LIN {X -112.034,Y -13.899,Z -33.351,A -90.000,B 90.000,C 0.000} C_DIS
LIN {X -111.882,Y -13.901,Z -33.215,A -90.000,B 90.000,C 0.000} C_DIS
LIN {X -111.725,Y -13.904,Z -33.072,A -90.000,B 90.000,C 0.000} C_DIS
LIN {X -111.571,Y -13.911,Z -32.939,A -90.000,B 90.000,C 0.000} C_DIS
LIN {X -111.426,Y -13.925,Z -32.809,A -90.000,B 90.000,C 0.000} C_DIS
LIN {X -111.312,Y -13.944,Z -32.695,A -90.000,B 90.000,C 0.000} C_DIS
LIN {X -110.883,Y -13.954,Z -32.137,A -90.000,B 90.000,C 0.000} C_DIS
LIN {X -110.737,Y -13.959,Z -31.950,A -90.000,B 90.000,C 0.000} C_DIS
LIN {X -110.627,Y -13.962,Z -31.815,A -90.000,B 90.000,C 0.000} C_DIS
LIN {X -110.356,Y -13.969,Z -31.490,A -90.000,B 90.000,C 0.000} C_DIS
LIN {X -110.187,Y -13.968,Z -31.297,A -90.000,B 90.000,C 0.000} C_DIS
LIN {X -110.090,Y -13.970,Z -31.191,A -90.000,B 90.000,C 0.000} C_DIS
LIN {X -109.713,Y -13.983,Z -30.801,A -90.000,B 90.000,C 0.000} C_DIS
LIN {X -109.313,Y -13.994,Z -30.426,A -90.000,B 90.000,C 0.000} C_DIS
LIN {X -108.942,Y -13.995,Z -30.095,A -90.000,B 90.000,C 0.000} C_DIS
LIN {X -108.599,Y -14.004,Z -29.802,A -90.000,B 90.000,C 0.000} C_DIS
LIN {X -108.444,Y -14.007,Z -29.672,A -90.000,B 90.000,C 0.000} C_DIS
LIN {X -108.225,Y -14.011,Z -29.494,A -90.000,B 90.000,C 0.000} C_DIS
LIN {X -107.679,Y -14.018,Z -29.057,A -90.000,B 90.000,C 0.000} C_DIS
LIN {X -107.487,Y -14.013,Z -28.912,A -90.000,B 90.000,C 0.000} C_DIS
LIN {X -107.181,Y -14.012,Z -28.694,A -90.000,B 90.000,C 0.000} C_DIS
LIN {X -106.850,Y -14.010,Z -28.465,A -90.000,B 90.000,C 0.000} C_DIS
LIN {X -106.554,Y -13.995,Z -28.277,A -90.000,B 90.000,C 0.000} C_DIS
LIN {X -106.262,Y -13.993,Z -28.107,A -90.000,B 90.000,C 0.000} C_DIS
LIN {X -105.912,Y -13.982,Z -27.915,A -90.000,B 90.000,C 0.000} C_DIS
LIN {X -105.604,Y -13.971,Z -27.766,A -90.000,B 90.000,C 0.000} C_DIS
LIN {X -105.412,Y -13.966,Z -27.676,A -90.000,B 90.000,C 0.000} C_DIS
LIN {X -105.178,Y -13.965,Z -27.574,A -90.000,B 90.000,C 0.000} C_DIS
LIN {X -104.756,Y -13.950,Z -27.404,A -90.000,B 90.000,C 0.000} C_DIS
LIN {X -104.528,Y -13.941,Z -27.320,A -90.000,B 90.000,C 0.000} C_DIS
LIN {X -104.102,Y -13.933,Z -27.170,A -90.000,B 90.000,C 0.000} C_DIS
LIN {X -103.873,Y -13.933,Z -27.095,A -90.000,B 90.000,C 0.000} C_DIS
LIN {X -103.252,Y -13.916,Z -26.894,A -90.000,B 90.000,C 0.000} C_DIS
LIN {X -102.946,Y -13.913,Z -26.800,A -90.000,B 90.000,C 0.000} C_DIS
LIN {X -102.732,Y -13.819,Z -26.639,A -90.000,B 90.000,C 0.000} C_DIS
LIN {X -102.589,Y -13.762,Z -26.537,A -90.000,B 90.000,C 0.000} C_DIS
LIN {X -102.458,Y -13.716,Z -26.450,A -90.000,B 90.000,C 0.000} C_DIS
LIN {X -102.318,Y -13.669,Z -26.360,A -90.000,B 90.000,C 0.000} C_DIS
LIN {X -102.306,Y -13.670,Z -26.341,A -90.000,B 90.000,C 0.000} C_DIS
LIN {X -102.042,Y -13.676,Z -25.951,A -90.000,B 90.000,C 0.000} C_DIS
LIN {X -101.875,Y -13.681,Z -25.720,A -90.000,B 90.000,C 0.000} C_DIS
LIN {X -101.706,Y -13.682,Z -25.502,A -90.000,B 90.000,C 0.000} C_DIS
LIN {X -101.671,Y -13.685,Z -25.450,A -90.000,B 90.000,C 0.000} C_DIS
LIN {X -101.467,Y -13.684,Z -25.192,A -90.000,B 90.000,C 0.000} C_DIS
LIN {X -101.393,Y -13.692,Z -25.087,A -90.000,B 90.000,C 0.000} C_DIS
LIN {X -101.277,Y -13.697,Z -24.936,A -90.000,B 90.000,C 0.000} C_DIS
LIN {X -101.079,Y -13.713,Z -24.676,A -90.000,B 90.000,C 0.000} C_DIS
LIN {X -100.863,Y -13.726,Z -24.406,A -90.000,B 90.000,C 0.000} C_DIS
LIN {X -100.744,Y -13.738,Z -24.262,A -90.000,B 90.000,C 0.000} C_DIS
LIN {X -100.655,Y -13.743,Z -24.163,A -90.000,B 90.000,C 0.000} C_DIS
LIN {X -100.615,Y -13.744,Z -24.116,A -90.000,B 90.000,C 0.000} C_DIS
LIN {X -100.507,Y -13.750,Z -23.996,A -90.000,B 90.000,C 0.000} C_DIS
LIN {X -100.359,Y -13.763,Z -23.838,A -90.000,B 90.000,C 0.000} C_DIS
LIN {X -100.223,Y -13.773,Z -23.695,A -90.000,B 90.000,C 0.000} C_DIS
LIN {X -99.934,Y -13.779,Z -23.429,A -90.000,B 90.000,C 0.000} C_DIS
LIN {X -99.843,Y -13.783,Z -23.348,A -90.000,B 90.000,C 0.000} C_DIS
LIN {X -99.649,Y -13.788,Z -23.183,A -90.000,B 90.000,C 0.000} C_DIS
LIN {X -99.518,Y -13.792,Z -23.082,A -90.000,B 90.000,C 0.000} C_DIS
LIN {X -99.172,Y -13.792,Z -22.838,A -90.000,B 90.000,C 0.000} C_DIS
LIN {X -98.955,Y -13.787,Z -22.696,A -90.000,B 90.000,C 0.000} C_DIS
LIN {X -98.690,Y -13.777,Z -22.542,A -90.000,B 90.000,C 0.000} C_DIS
LIN {X -98.581,Y -13.777,Z -22.483,A -90.000,B 90.000,C 0.000} C_DIS
LIN {X -98.305,Y -13.760,Z -22.357,A -90.000,B 90.000,C 0.000} C_DIS
LIN {X -98.201,Y -13.756,Z -22.312,A -90.000,B 90.000,C 0.000} C_DIS
LIN {X -98.005,Y -13.745,Z -22.237,A -90.000,B 90.000,C 0.000} C_DIS
LIN {X -97.903,Y -13.741,Z -22.200,A -90.000,B 90.000,C 0.000} C_DIS
LIN {X -97.496,Y -13.717,Z -22.072,A -90.000,B 90.000,C 0.000} C_DIS
LIN {X -97.397,Y -13.709,Z -22.050,A -90.000,B 90.000,C 0.000} C_DIS
LIN {X -97.037,Y -13.687,Z -21.979,A -90.000,B 90.000,C 0.000} C_DIS
LIN {X -96.920,Y -13.678,Z -21.961,A -90.000,B 90.000,C 0.000} C_DIS
LIN {X -96.713,Y -13.661,Z -21.934,A -90.000,B 90.000,C 0.000} C_DIS
LIN {X -96.487,Y -13.648,Z -21.909,A -90.000,B 90.000,C 0.000} C_DIS
LIN {X -96.193,Y -13.619,Z -21.899,A -90.000,B 90.000,C 0.000} C_DIS
LIN {X -96.028,Y -13.611,Z -21.893,A -90.000,B 90.000,C 0.000} C_DIS
LIN {X -95.877,Y -13.604,Z -21.893,A -90.000,B 90.000,C 0.000} C_DIS
LIN {X -95.614,Y -13.584,Z -21.906,A -90.000,B 90.000,C 0.000} C_DIS
LIN {X -95.537,Y -13.622,Z -21.843,A -90.000,B 90.000,C 0.000} C_DIS
LIN {X -95.434,Y -13.674,Z -21.767,A -90.000,B 90.000,C 0.000} C_DIS
LIN {X -95.337,Y -13.724,Z -21.703,A -90.000,B 90.000,C 0.000} C_DIS
LIN {X -95.205,Y -13.792,Z -21.624,A -90.000,B 90.000,C 0.000} C_DIS
LIN {X -95.067,Y -13.866,Z -21.548,A -90.000,B 90.000,C 0.000} C_DIS
LIN {X -94.996,Y -13.904,Z -21.514,A -90.000,B 90.000,C 0.000} C_DIS
LIN {X -94.934,Y -13.938,Z -21.487,A -90.000,B 90.000,C 0.000} C_DIS
LIN {X -94.872,Y -13.972,Z -21.461,A -90.000,B 90.000,C 0.000} C_DIS
LIN {X -94.732,Y -14.044,Z -21.414,A -90.000,B 90.000,C 0.000} C_DIS
LIN {X -94.570,Y -14.126,Z -21.368,A -90.000,B 90.000,C 0.000} C_DIS
LIN {X -94.236,Y -14.315,Z -21.280,A -90.000,B 90.000,C 0.000} C_DIS
LIN {X -94.158,Y -14.359,Z -21.266,A -90.000,B 90.000,C 0.000} C_DIS
LIN {X -94.070,Y -14.402,Z -21.258,A -90.000,B 90.000,C 0.000} C_DIS
LIN {X -93.862,Y -14.506,Z -21.250,A -90.000,B 90.000,C 0.000} C_DIS
LIN {X -93.860,Y -14.506,Z -21.241,A -90.000,B 90.000,C 0.000} C_DIS
LIN {X -93.780,Y -14.481,Z -20.924,A -90.000,B 90.000,C 0.000} C_DIS
LIN {X -93.747,Y -14.467,Z -20.815,A -90.000,B 90.000,C 0.000} C_DIS
LIN {X -93.701,Y -14.454,Z -20.689,A -90.000,B 90.000,C 0.000} C_DIS
LIN {X -93.679,Y -14.449,Z -20.634,A -90.000,B 90.000,C 0.000} C_DIS
LIN {X -93.611,Y -14.437,Z -20.486,A -90.000,B 90.000,C 0.000} C_DIS
LIN {X -93.534,Y -14.428,Z -20.316,A -90.000,B 90.000,C 0.000} C_DIS
LIN {X -93.448,Y -14.408,Z -20.153,A -90.000,B 90.000,C 0.000} C_DIS
LIN {X -93.387,Y -14.400,Z -20.053,A -90.000,B 90.000,C 0.000} C_DIS
LIN {X -93.227,Y -14.381,Z -19.822,A -90.000,B 90.000,C 0.000} C_DIS
LIN {X -93.122,Y -14.364,Z -19.684,A -90.000,B 90.000,C 0.000} C_DIS
LIN {X -93.056,Y -14.356,Z -19.608,A -90.000,B 90.000,C 0.000} C_DIS
LIN {X -92.999,Y -14.351,Z -19.545,A -90.000,B 90.000,C 0.000} C_DIS
LIN {X -92.781,Y -14.328,Z -19.328,A -90.000,B 90.000,C 0.000} C_DIS
LIN {X -92.711,Y -14.319,Z -19.266,A -90.000,B 90.000,C 0.000} C_DIS
LIN {X -92.547,Y -14.302,Z -19.126,A -90.000,B 90.000,C 0.000} C_DIS
LIN {X -92.372,Y -14.279,Z -18.982,A -90.000,B 90.000,C 0.000} C_DIS
LIN {X -92.286,Y -14.270,Z -18.915,A -90.000,B 90.000,C 0.000} C_DIS
LIN {X -92.090,Y -14.252,Z -18.764,A -90.000,B 90.000,C 0.000} C_DIS
LIN {X -92.005,Y -14.240,Z -18.704,A -90.000,B 90.000,C 0.000} C_DIS
LIN {X -91.863,Y -14.227,Z -18.614,A -90.000,B 90.000,C 0.000} C_DIS
LIN {X -91.754,Y -14.219,Z -18.547,A -90.000,B 90.000,C 0.000} C_DIS
LIN {X -91.610,Y -14.201,Z -18.466,A -90.000,B 90.000,C 0.000} C_DIS
LIN {X -91.370,Y -14.176,Z -18.340,A -90.000,B 90.000,C 0.000} C_DIS
LIN {X -91.178,Y -14.158,Z -18.248,A -90.000,B 90.000,C 0.000} C_DIS
LIN {X -91.044,Y -14.151,Z -18.189,A -90.000,B 90.000,C 0.000} C_DIS
LIN {X -90.692,Y -14.145,Z -18.053,A -90.000,B 90.000,C 0.000} C_DIS
LIN {X -90.538,Y -14.145,Z -18.001,A -90.000,B 90.000,C 0.000} C_DIS
LIN {X -90.152,Y -14.128,Z -17.893,A -90.000,B 90.000,C 0.000} C_DIS
LIN {X -89.604,Y -14.082,Z -17.756,A -90.000,B 90.000,C 0.000} C_DIS
LIN {X -89.384,Y -14.072,Z -17.709,A -90.000,B 90.000,C 0.000} C_DIS
LIN {X -89.128,Y -14.063,Z -17.660,A -90.000,B 90.000,C 0.000} C_DIS
LIN {X -88.983,Y -14.061,Z -17.638,A -90.000,B 90.000,C 0.000} C_DIS
LIN {X -88.897,Y -14.064,Z -17.628,A -90.000,B 90.000,C 0.000} C_DIS
LIN {X -88.803,Y -14.066,Z -17.620,A -90.000,B 90.000,C 0.000} C_DIS
LIN {X -88.585,Y -14.060,Z -17.609,A -90.000,B 90.000,C 0.000} C_DIS
LIN {X -88.469,Y -14.059,Z -17.606,A -90.000,B 90.000,C 0.000} C_DIS
LIN {X -87.435,Y -14.047,Z -17.615,A -90.000,B 90.000,C 0.000} C_DIS
LIN {X -87.313,Y -14.047,Z -17.617,A -90.000,B 90.000,C 0.000} C_DIS
LIN {X -86.918,Y -14.044,Z -17.651,A -90.000,B 90.000,C 0.000} C_DIS
LIN {X -86.812,Y -14.039,Z -17.668,A -90.000,B 90.000,C 0.000} C_DIS
LIN {X -86.741,Y -14.038,Z -17.683,A -90.000,B 90.000,C 0.000} C_DIS
LIN {X -86.721,Y -14.022,Z -17.671,A -90.000,B 90.000,C 0.000} C_DIS
LIN {X -86.608,Y -13.934,Z -17.624,A -90.000,B 90.000,C 0.000} C_DIS
LIN {X -86.542,Y -13.886,Z -17.598,A -90.000,B 90.000,C 0.000} C_DIS
LIN {X -86.312,Y -13.734,Z -17.528,A -90.000,B 90.000,C 0.000} C_DIS
LIN {X -86.280,Y -13.716,Z -17.521,A -90.000,B 90.000,C 0.000} C_DIS
LIN {X -86.235,Y -13.716,Z -17.433,A -90.000,B 90.000,C 0.000} C_DIS
LIN {X -86.137,Y -13.714,Z -17.283,A -90.000,B 90.000,C 0.000} C_DIS
LIN {X -85.985,Y -13.712,Z -17.053,A -90.000,B 90.000,C 0.000} C_DIS
LIN {X -85.847,Y -13.708,Z -16.857,A -90.000,B 90.000,C 0.000} C_DIS
LIN {X -85.774,Y -13.702,Z -16.762,A -90.000,B 90.000,C 0.000} C_DIS
LIN {X -85.680,Y -13.698,Z -16.647,A -90.000,B 90.000,C 0.000} C_DIS
LIN {X -85.521,Y -13.698,Z -16.460,A -90.000,B 90.000,C 0.000} C_DIS
LIN {X -85.383,Y -13.687,Z -16.321,A -90.000,B 90.000,C 0.000} C_DIS
LIN {X -85.294,Y -13.683,Z -16.234,A -90.000,B 90.000,C 0.000} C_DIS
LIN {X -85.213,Y -13.682,Z -16.157,A -90.000,B 90.000,C 0.000} C_DIS
LIN {X -85.158,Y -13.679,Z -16.108,A -90.000,B 90.000,C 0.000} C_DIS
LIN {X -84.818,Y -13.662,Z -15.820,A -90.000,B 90.000,C 0.000} C_DIS
LIN {X -84.702,Y -13.654,Z -15.727,A -90.000,B 90.000,C 0.000} C_DIS
LIN {X -84.628,Y -13.649,Z -15.671,A -90.000,B 90.000,C 0.000} C_DIS
LIN {X -84.520,Y -13.646,Z -15.593,A -90.000,B 90.000,C 0.000} C_DIS
LIN {X -84.262,Y -13.636,Z -15.421,A -90.000,B 90.000,C 0.000} C_DIS
LIN {X -84.126,Y -13.632,Z -15.333,A -90.000,B 90.000,C 0.000} C_DIS
LIN {X -83.745,Y -13.611,Z -15.131,A -90.000,B 90.000,C 0.000} C_DIS
LIN {X -83.301,Y -13.590,Z -14.916,A -90.000,B 90.000,C 0.000} C_DIS
LIN {X -83.060,Y -13.582,Z -14.816,A -90.000,B 90.000,C 0.000} C_DIS
LIN {X -82.848,Y -13.572,Z -14.733,A -90.000,B 90.000,C 0.000} C_DIS
LIN {X -82.617,Y -13.562,Z -14.656,A -90.000,B 90.000,C 0.000} C_DIS
LIN {X -82.394,Y -13.551,Z -14.586,A -90.000,B 90.000,C 0.000} C_DIS
LIN {X -82.185,Y -13.542,Z -14.524,A -90.000,B 90.000,C 0.000} C_DIS
LIN {X -81.813,Y -13.532,Z -14.411,A -90.000,B 90.000,C 0.000} C_DIS
LIN {X -81.344,Y -13.519,Z -14.313,A -90.000,B 90.000,C 0.000} C_DIS
LIN {X -81.190,Y -13.515,Z -14.281,A -90.000,B 90.000,C 0.000} C_DIS
LIN {X -80.857,Y -13.504,Z -14.223,A -90.000,B 90.000,C 0.000} C_DIS
LIN {X -80.728,Y -13.500,Z -14.198,A -90.000,B 90.000,C 0.000} C_DIS
LIN {X -80.638,Y -13.500,Z -14.182,A -90.000,B 90.000,C 0.000} C_DIS
LIN {X -80.232,Y -13.495,Z -14.137,A -90.000,B 90.000,C 0.000} C_DIS
LIN {X -80.019,Y -13.494,Z -14.111,A -90.000,B 90.000,C 0.000} C_DIS
LIN {X -79.547,Y -13.485,Z -14.066,A -90.000,B 90.000,C 0.000} C_DIS
LIN {X -79.213,Y -13.482,Z -14.039,A -90.000,B 90.000,C 0.000} C_DIS
LIN {X -79.139,Y -13.481,Z -14.037,A -90.000,B 90.000,C 0.000} C_DIS
LIN {X -78.717,Y -13.481,Z -14.026,A -90.000,B 90.000,C 0.000} C_DIS
LIN {X -78.513,Y -13.479,Z -14.025,A -90.000,B 90.000,C 0.000} C_DIS
LIN {X -78.013,Y -13.473,Z -14.031,A -90.000,B 90.000,C 0.000} C_DIS
LIN {X -77.640,Y -13.471,Z -14.042,A -90.000,B 90.000,C 0.000} C_DIS
LIN {X -77.520,Y -13.469,Z -14.050,A -90.000,B 90.000,C 0.000} C_DIS
LIN {X -77.155,Y -13.472,Z -14.080,A -90.000,B 90.000,C 0.000} C_DIS
LIN {X -76.920,Y -13.471,Z -14.109,A -90.000,B 90.000,C 0.000} C_DIS
LIN {X -76.442,Y -13.464,Z -14.180,A -90.000,B 90.000,C 0.000} C_DIS
LIN {X -76.162,Y -13.461,Z -14.224,A -90.000,B 90.000,C 0.000} C_DIS
LIN {X -75.940,Y -13.459,Z -14.264,A -90.000,B 90.000,C 0.000} C_DIS
LIN {X -75.365,Y -13.465,Z -14.380,A -90.000,B 90.000,C 0.000} C_DIS
LIN {X -74.909,Y -13.460,Z -14.500,A -90.000,B 90.000,C 0.000} C_DIS
LIN {X -74.580,Y -13.456,Z -14.593,A -90.000,B 90.000,C 0.000} C_DIS
LIN {X -74.366,Y -13.450,Z -14.663,A -90.000,B 90.000,C 0.000} C_DIS
LIN {X -74.120,Y -13.447,Z -14.745,A -90.000,B 90.000,C 0.000} C_DIS
LIN {X -73.815,Y -13.449,Z -14.848,A -90.000,B 90.000,C 0.000} C_DIS
LIN {X -72.971,Y -13.458,Z -15.136,A -90.000,B 90.000,C 0.000} C_DIS
LIN {X -72.702,Y -13.458,Z -15.238,A -90.000,B 90.000,C 0.000} C_DIS
LIN {X -72.379,Y -13.457,Z -15.363,A -90.000,B 90.000,C 0.000} C_DIS
LIN {X -72.204,Y -13.451,Z -15.444,A -90.000,B 90.000,C 0.000} C_DIS
LIN {X -71.892,Y -13.451,Z -15.592,A -90.000,B 90.000,C 0.000} C_DIS
LIN {X -71.809,Y -13.451,Z -15.631,A -90.000,B 90.000,C 0.000} C_DIS
LIN {X -70.378,Y -13.450,Z -16.339,A -90.000,B 90.000,C 0.000} C_DIS
LIN {X -69.618,Y -13.460,Z -16.736,A -90.000,B 90.000,C 0.000} C_DIS
LIN {X -68.763,Y -13.469,Z -17.184,A -90.000,B 90.000,C 0.000} C_DIS
LIN {X -67.645,Y -13.489,Z -17.780,A -90.000,B 90.000,C 0.000} C_DIS
LIN {X -67.198,Y -13.496,Z -18.025,A -90.000,B 90.000,C 0.000} C_DIS
LIN {X -66.565,Y -13.511,Z -18.361,A -90.000,B 90.000,C 0.000} C_DIS
LIN {X -65.801,Y -13.530,Z -18.795,A -90.000,B 90.000,C 0.000} C_DIS
LIN {X -65.574,Y -13.544,Z -18.914,A -90.000,B 90.000,C 0.000} C_DIS
LIN {X -65.396,Y -13.551,Z -19.018,A -90.000,B 90.000,C 0.000} C_DIS
LIN {X -64.571,Y -13.586,Z -19.501,A -90.000,B 90.000,C 0.000} C_DIS
LIN {X -64.308,Y -13.607,Z -19.641,A -90.000,B 90.000,C 0.000} C_DIS
LIN {X -63.999,Y -13.623,Z -19.825,A -90.000,B 90.000,C 0.000} C_DIS
LIN {X -63.495,Y -13.656,Z -20.131,A -90.000,B 90.000,C 0.000} C_DIS
LIN {X -63.469,Y -13.659,Z -20.145,A -90.000,B 90.000,C 0.000} C_DIS
LIN {X -62.802,Y -13.710,Z -20.544,A -90.000,B 90.000,C 0.000} C_DIS
LIN {X -62.463,Y -13.736,Z -20.756,A -90.000,B 90.000,C 0.000} C_DIS
LIN {X -62.354,Y -13.749,Z -20.815,A -90.000,B 90.000,C 0.000} C_DIS
LIN {X -62.041,Y -13.777,Z -21.008,A -90.000,B 90.000,C 0.000} C_DIS
LIN {X -61.752,Y -13.808,Z -21.196,A -90.000,B 90.000,C 0.000} C_DIS
LIN {X -61.442,Y -13.831,Z -21.391,A -90.000,B 90.000,C 0.000} C_DIS
LIN {X -60.969,Y -13.887,Z -21.668,A -90.000,B 90.000,C 0.000} C_DIS
LIN {X -60.722,Y -13.907,Z -21.825,A -90.000,B 90.000,C 0.000} C_DIS
LIN {X -60.550,Y -13.917,Z -21.930,A -90.000,B 90.000,C 0.000} C_DIS
LIN {X -60.491,Y -13.924,Z -21.963,A -90.000,B 90.000,C 0.000} C_DIS
LIN {X -60.176,Y -13.953,Z -22.144,A -90.000,B 90.000,C 0.000} C_DIS
LIN {X -59.949,Y -13.961,Z -22.261,A -90.000,B 90.000,C 0.000} C_DIS
LIN {X -59.647,Y -13.971,Z -22.420,A -90.000,B 90.000,C 0.000} C_DIS
LIN {X -59.462,Y -13.985,Z -22.509,A -90.000,B 90.000,C 0.000} C_DIS
LIN {X -59.050,Y -13.997,Z -22.683,A -90.000,B 90.000,C 0.000} C_DIS
LIN {X -58.693,Y -14.004,Z -22.838,A -90.000,B 90.000,C 0.000} C_DIS
LIN {X -58.569,Y -14.009,Z -22.888,A -90.000,B 90.000,C 0.000} C_DIS
LIN {X -57.557,Y -14.022,Z -23.247,A -90.000,B 90.000,C 0.000} C_DIS
LIN {X -57.259,Y -14.023,Z -23.356,A -90.000,B 90.000,C 0.000} C_DIS
LIN {X -57.092,Y -14.023,Z -23.408,A -90.000,B 90.000,C 0.000} C_DIS
LIN {X -56.518,Y -14.030,Z -23.584,A -90.000,B 90.000,C 0.000} C_DIS
LIN {X -55.731,Y -14.034,Z -23.819,A -90.000,B 90.000,C 0.000} C_DIS
LIN {X -55.658,Y -14.033,Z -23.840,A -90.000,B 90.000,C 0.000} C_DIS
LIN {X -55.037,Y -14.036,Z -24.006,A -90.000,B 90.000,C 0.000} C_DIS
LIN {X -54.393,Y -14.033,Z -24.173,A -90.000,B 90.000,C 0.000} C_DIS
LIN {X -54.063,Y -14.037,Z -24.253,A -90.000,B 90.000,C 0.000} C_DIS
LIN {X -53.491,Y -14.045,Z -24.391,A -90.000,B 90.000,C 0.000} C_DIS
LIN {X -53.098,Y -14.047,Z -24.472,A -90.000,B 90.000,C 0.000} C_DIS
LIN {X -51.762,Y -14.064,Z -24.759,A -90.000,B 90.000,C 0.000} C_DIS
LIN {X -51.233,Y -14.065,Z -24.866,A -90.000,B 90.000,C 0.000} C_DIS
LIN {X -50.477,Y -14.068,Z -25.002,A -90.000,B 90.000,C 0.000} C_DIS
LIN {X -49.024,Y -14.058,Z -25.239,A -90.000,B 90.000,C 0.000} C_DIS
LIN {X -48.480,Y -14.057,Z -25.331,A -90.000,B 90.000,C 0.000} C_DIS
LIN {X -47.532,Y -14.044,Z -25.471,A -90.000,B 90.000,C 0.000} C_DIS
LIN {X -46.298,Y -14.022,Z -25.659,A -90.000,B 90.000,C 0.000} C_DIS
LIN {X -45.477,Y -13.997,Z -25.792,A -90.000,B 90.000,C 0.000} C_DIS
LIN {X -44.914,Y -13.987,Z -25.889,A -90.000,B 90.000,C 0.000} C_DIS
LIN {X -44.631,Y -13.982,Z -25.935,A -90.000,B 90.000,C 0.000} C_DIS
LIN {X -44.518,Y -13.978,Z -25.955,A -90.000,B 90.000,C 0.000} C_DIS
LIN {X -43.197,Y -13.938,Z -26.189,A -90.000,B 90.000,C 0.000} C_DIS
LIN {X -42.434,Y -13.912,Z -26.327,A -90.000,B 90.000,C 0.000} C_DIS
LIN {X -41.770,Y -13.897,Z -26.456,A -90.000,B 90.000,C 0.000} C_DIS
LIN {X -41.004,Y -13.874,Z -26.611,A -90.000,B 90.000,C 0.000} C_DIS
LIN {X -40.551,Y -13.859,Z -26.698,A -90.000,B 90.000,C 0.000} C_DIS
LIN {X -39.970,Y -13.847,Z -26.814,A -90.000,B 90.000,C 0.000} C_DIS
LIN {X -38.902,Y -13.819,Z -27.052,A -90.000,B 90.000,C 0.000} C_DIS
LIN {X -38.244,Y -13.808,Z -27.195,A -90.000,B 90.000,C 0.000} C_DIS
LIN {X -37.854,Y -13.799,Z -27.283,A -90.000,B 90.000,C 0.000} C_DIS
LIN {X -37.466,Y -13.793,Z -27.374,A -90.000,B 90.000,C 0.000} C_DIS
LIN {X -36.421,Y -13.777,Z -27.608,A -90.000,B 90.000,C 0.000} C_DIS
LIN {X -36.023,Y -13.769,Z -27.700,A -90.000,B 90.000,C 0.000} C_DIS
LIN {X -35.198,Y -13.758,Z -27.895,A -90.000,B 90.000,C 0.000} C_DIS
LIN {X -34.304,Y -13.755,Z -28.099,A -90.000,B 90.000,C 0.000} C_DIS
LIN {X -34.187,Y -13.763,Z -28.116,A -90.000,B 90.000,C 0.000} C_DIS
LIN {X -32.560,Y -13.874,Z -28.356,A -90.000,B 90.000,C 0.000} C_DIS
LIN {X -31.936,Y -13.923,Z -28.446,A -90.000,B 90.000,C 0.000} C_DIS
LIN {X -31.312,Y -13.969,Z -28.544,A -90.000,B 90.000,C 0.000} C_DIS
LIN {X -30.091,Y -14.060,Z -28.739,A -90.000,B 90.000,C 0.000} C_DIS
LIN {X -28.790,Y -14.155,Z -28.954,A -90.000,B 90.000,C 0.000} C_DIS
LIN {X -28.283,Y -14.189,Z -29.029,A -90.000,B 90.000,C 0.000} C_DIS
LIN {X -27.818,Y -14.222,Z -29.095,A -90.000,B 90.000,C 0.000} C_DIS
LIN {X -26.794,Y -14.282,Z -29.244,A -90.000,B 90.000,C 0.000} C_DIS
LIN {X -26.640,Y -14.289,Z -29.265,A -90.000,B 90.000,C 0.000} C_DIS
LIN {X -26.107,Y -14.309,Z -29.323,A -90.000,B 90.000,C 0.000} C_DIS
LIN {X -25.922,Y -14.312,Z -29.337,A -90.000,B 90.000,C 0.000} C_DIS
LIN {X -25.484,Y -14.324,Z -29.368,A -90.000,B 90.000,C 0.000} C_DIS
LIN {X -25.205,Y -14.319,Z -29.378,A -90.000,B 90.000,C 0.000} C_DIS
LIN {X -24.830,Y -14.312,Z -29.398,A -90.000,B 90.000,C 0.000} C_DIS
LIN {X -24.748,Y -14.307,Z -29.398,A -90.000,B 90.000,C 0.000} C_DIS
LIN {X -24.057,Y -14.271,Z -29.410,A -90.000,B 90.000,C 0.000} C_DIS
LIN {X -23.493,Y -14.250,Z -29.433,A -90.000,B 90.000,C 0.000} C_DIS
LIN {X -23.250,Y -14.237,Z -29.444,A -90.000,B 90.000,C 0.000} C_DIS
LIN {X -22.902,Y -14.213,Z -29.462,A -90.000,B 90.000,C 0.000} C_DIS
LIN {X -22.417,Y -14.190,Z -29.501,A -90.000,B 90.000,C 0.000} C_DIS
LIN {X -21.725,Y -14.162,Z -29.559,A -90.000,B 90.000,C 0.000} C_DIS
LIN {X -21.512,Y -14.150,Z -29.580,A -90.000,B 90.000,C 0.000} C_DIS
LIN {X -21.132,Y -14.134,Z -29.621,A -90.000,B 90.000,C 0.000} C_DIS
LIN {X -19.896,Y -14.096,Z -29.773,A -90.000,B 90.000,C 0.000} C_DIS
LIN {X -18.994,Y -14.069,Z -29.888,A -90.000,B 90.000,C 0.000} C_DIS
LIN {X -18.061,Y -14.046,Z -30.019,A -90.000,B 90.000,C 0.000} C_DIS
LIN {X -16.881,Y -14.026,Z -30.201,A -90.000,B 90.000,C 0.000} C_DIS
LIN {X -16.404,Y -14.009,Z -30.283,A -90.000,B 90.000,C 0.000} C_DIS
LIN {X -15.575,Y -13.995,Z -30.441,A -90.000,B 90.000,C 0.000} C_DIS
LIN {X -15.024,Y -13.986,Z -30.548,A -90.000,B 90.000,C 0.000} C_DIS
LIN {X -13.431,Y -13.971,Z -30.881,A -90.000,B 90.000,C 0.000} C_DIS
LIN {X -13.324,Y -13.971,Z -30.902,A -90.000,B 90.000,C 0.000} C_DIS
LIN {X -12.405,Y -13.961,Z -31.070,A -90.000,B 90.000,C 0.000} C_DIS
LIN {X -12.011,Y -13.956,Z -31.148,A -90.000,B 90.000,C 0.000} C_DIS
LIN {X -11.638,Y -13.954,Z -31.226,A -90.000,B 90.000,C 0.000} C_DIS
LIN {X -11.400,Y -13.947,Z -31.271,A -90.000,B 90.000,C 0.000} C_DIS
LIN {X -10.523,Y -13.938,Z -31.421,A -90.000,B 90.000,C 0.000} C_DIS
LIN {X -9.659,Y -13.938,Z -31.578,A -90.000,B 90.000,C 0.000} C_DIS
LIN {X -9.259,Y -13.937,Z -31.652,A -90.000,B 90.000,C 0.000} C_DIS
LIN {X -8.758,Y -13.939,Z -31.740,A -90.000,B 90.000,C 0.000} C_DIS
LIN {X -8.129,Y -13.937,Z -31.856,A -90.000,B 90.000,C 0.000} C_DIS
LIN {X -6.693,Y -13.948,Z -32.138,A -90.000,B 90.000,C 0.000} C_DIS
LIN {X -6.485,Y -13.947,Z -32.175,A -90.000,B 90.000,C 0.000} C_DIS
LIN {X -6.144,Y -13.941,Z -32.237,A -90.000,B 90.000,C 0.000} C_DIS
LIN {X -4.545,Y -13.932,Z -32.541,A -90.000,B 90.000,C 0.000} C_DIS
LIN {X -3.564,Y -13.908,Z -32.712,A -90.000,B 90.000,C 0.000} C_DIS
LIN {X -1.900,Y -13.868,Z -32.979,A -90.000,B 90.000,C 0.000} C_DIS
LIN {X -0.666,Y -13.854,Z -33.160,A -90.000,B 90.000,C 0.000} C_DIS
LIN {X 0.364,Y -13.835,Z -33.320,A -90.000,B 90.000,C 0.000} C_DIS
LIN {X 0.630,Y -13.835,Z -33.359,A -90.000,B 90.000,C 0.000} C_DIS
LIN {X 2.120,Y -13.844,Z -33.588,A -90.000,B 90.000,C 0.000} C_DIS
LIN {X 2.655,Y -13.842,Z -33.679,A -90.000,B 90.000,C 0.000} C_DIS
LIN {X 3.036,Y -13.845,Z -33.741,A -90.000,B 90.000,C 0.000} C_DIS
LIN {X 4.469,Y -13.858,Z -33.974,A -90.000,B 90.000,C 0.000} C_DIS
LIN {X 4.778,Y -13.859,Z -34.022,A -90.000,B 90.000,C 0.000} C_DIS
LIN {X 5.606,Y -13.863,Z -34.174,A -90.000,B 90.000,C 0.000} C_DIS
LIN {X 6.682,Y -13.857,Z -34.382,A -90.000,B 90.000,C 0.000} C_DIS
LIN {X 7.507,Y -13.849,Z -34.538,A -90.000,B 90.000,C 0.000} C_DIS
LIN {X 8.033,Y -13.848,Z -34.654,A -90.000,B 90.000,C 0.000} C_DIS
LIN {X 10.011,Y -13.831,Z -35.104,A -90.000,B 90.000,C 0.000} C_DIS
LIN {X 10.789,Y -13.829,Z -35.289,A -90.000,B 90.000,C 0.000} C_DIS
LIN {X 11.350,Y -13.826,Z -35.426,A -90.000,B 90.000,C 0.000} C_DIS
LIN {X 12.489,Y -13.812,Z -35.696,A -90.000,B 90.000,C 0.000} C_DIS
LIN {X 13.654,Y -13.807,Z -35.961,A -90.000,B 90.000,C 0.000} C_DIS
LIN {X 14.337,Y -13.798,Z -36.111,A -90.000,B 90.000,C 0.000} C_DIS
LIN {X 14.558,Y -13.800,Z -36.154,A -90.000,B 90.000,C 0.000} C_DIS
LIN {X 14.947,Y -13.798,Z -36.222,A -90.000,B 90.000,C 0.000} C_DIS
LIN {X 15.730,Y -13.799,Z -36.355,A -90.000,B 90.000,C 0.000} C_DIS
LIN {X 16.108,Y -13.794,Z -36.415,A -90.000,B 90.000,C 0.000} C_DIS
LIN {X 16.238,Y -13.799,Z -36.429,A -90.000,B 90.000,C 0.000} C_DIS
LIN {X 16.404,Y -13.805,Z -36.446,A -90.000,B 90.000,C 0.000} C_DIS
LIN {X 16.528,Y -13.812,Z -36.456,A -90.000,B 90.000,C 0.000} C_DIS
LIN {X 17.228,Y -13.820,Z -36.484,A -90.000,B 90.000,C 0.000} C_DIS
LIN {X 17.549,Y -13.811,Z -36.486,A -90.000,B 90.000,C 0.000} C_DIS
LIN {X 17.799,Y -13.818,Z -36.472,A -90.000,B 90.000,C 0.000} C_DIS
LIN {X 18.097,Y -13.824,Z -36.453,A -90.000,B 90.000,C 0.000} C_DIS
LIN {X 18.543,Y -13.819,Z -36.412,A -90.000,B 90.000,C 0.000} C_DIS
LIN {X 18.690,Y -13.814,Z -36.401,A -90.000,B 90.000,C 0.000} C_DIS
LIN {X 18.731,Y -13.814,Z -36.396,A -90.000,B 90.000,C 0.000} C_DIS
LIN {X 19.607,Y -13.814,Z -36.323,A -90.000,B 90.000,C 0.000} C_DIS
LIN {X 19.814,Y -13.811,Z -36.303,A -90.000,B 90.000,C 0.000} C_DIS
LIN {X 20.174,Y -13.816,Z -36.257,A -90.000,B 90.000,C 0.000} C_DIS
LIN {X 20.788,Y -13.810,Z -36.193,A -90.000,B 90.000,C 0.000} C_DIS
LIN {X 21.155,Y -13.814,Z -36.147,A -90.000,B 90.000,C 0.000} C_DIS
LIN {X 21.648,Y -13.813,Z -36.100,A -90.000,B 90.000,C 0.000} C_DIS
LIN {X 21.858,Y -13.809,Z -36.084,A -90.000,B 90.000,C 0.000} C_DIS
LIN {X 22.208,Y -13.806,Z -36.061,A -90.000,B 90.000,C 0.000} C_DIS
LIN {X 22.816,Y -13.796,Z -36.030,A -90.000,B 90.000,C 0.000} C_DIS
LIN {X 23.146,Y -13.794,Z -36.016,A -90.000,B 90.000,C 0.000} C_DIS
LIN {X 23.504,Y -13.789,Z -36.007,A -90.000,B 90.000,C 0.000} C_DIS
LIN {X 24.314,Y -13.768,Z -35.991,A -90.000,B 90.000,C 0.000} C_DIS
LIN {X 24.960,Y -13.747,Z -35.991,A -90.000,B 90.000,C 0.000} C_DIS
LIN {X 25.413,Y -13.735,Z -35.989,A -90.000,B 90.000,C 0.000} C_DIS
LIN {X 25.835,Y -13.720,Z -35.995,A -90.000,B 90.000,C 0.000} C_DIS
LIN {X 26.233,Y -13.706,Z -36.002,A -90.000,B 90.000,C 0.000} C_DIS
LIN {X 26.583,Y -13.696,Z -36.011,A -90.000,B 90.000,C 0.000} C_DIS
LIN {X 27.555,Y -13.657,Z -36.048,A -90.000,B 90.000,C 0.000} C_DIS
LIN {X 27.739,Y -13.652,Z -36.058,A -90.000,B 90.000,C 0.000} C_DIS
LIN {X 28.255,Y -13.636,Z -36.095,A -90.000,B 90.000,C 0.000} C_DIS
LIN {X 28.934,Y -13.606,Z -36.146,A -90.000,B 90.000,C 0.000} C_DIS
LIN {X 29.228,Y -13.595,Z -36.166,A -90.000,B 90.000,C 0.000} C_DIS
LIN {X 30.080,Y -13.561,Z -36.238,A -90.000,B 90.000,C 0.000} C_DIS
LIN {X 30.564,Y -13.547,Z -36.280,A -90.000,B 90.000,C 0.000} C_DIS
LIN {X 31.181,Y -13.523,Z -36.346,A -90.000,B 90.000,C 0.000} C_DIS
LIN {X 31.673,Y -13.501,Z -36.397,A -90.000,B 90.000,C 0.000} C_DIS
LIN {X 32.315,Y -13.475,Z -36.465,A -90.000,B 90.000,C 0.000} C_DIS
LIN {X 32.680,Y -13.465,Z -36.500,A -90.000,B 90.000,C 0.000} C_DIS
LIN {X 33.128,Y -13.451,Z -36.551,A -90.000,B 90.000,C 0.000} C_DIS
LIN {X 34.364,Y -13.415,Z -36.701,A -90.000,B 90.000,C 0.000} C_DIS
LIN {X 34.841,Y -13.403,Z -36.770,A -90.000,B 90.000,C 0.000} C_DIS
LIN {X 35.286,Y -13.389,Z -36.843,A -90.000,B 90.000,C 0.000} C_DIS
LIN {X 35.853,Y -13.375,Z -36.925,A -90.000,B 90.000,C 0.000} C_DIS
LIN {X 36.309,Y -13.367,Z -37.002,A -90.000,B 90.000,C 0.000} C_DIS
LIN {X 37.253,Y -13.348,Z -37.179,A -90.000,B 90.000,C 0.000} C_DIS
LIN {X 37.764,Y -13.343,Z -37.275,A -90.000,B 90.000,C 0.000} C_DIS
LIN {X 38.133,Y -13.339,Z -37.350,A -90.000,B 90.000,C 0.000} C_DIS
LIN {X 38.405,Y -13.334,Z -37.421,A -90.000,B 90.000,C 0.000} C_DIS
LIN {X 38.992,Y -13.327,Z -37.559,A -90.000,B 90.000,C 0.000} C_DIS
LIN {X 40.071,Y -13.317,Z -37.820,A -90.000,B 90.000,C 0.000} C_DIS
LIN {X 40.816,Y -13.315,Z -38.002,A -90.000,B 90.000,C 0.000} C_DIS
LIN {X 41.263,Y -13.313,Z -38.135,A -90.000,B 90.000,C 0.000} C_DIS
LIN {X 41.839,Y -13.311,Z -38.318,A -90.000,B 90.000,C 0.000} C_DIS
LIN {X 43.350,Y -13.309,Z -38.757,A -90.000,B 90.000,C 0.000} C_DIS
LIN {X 43.882,Y -13.309,Z -38.915,A -90.000,B 90.000,C 0.000} C_DIS
LIN {X 44.676,Y -13.308,Z -39.193,A -90.000,B 90.000,C 0.000} C_DIS
LIN {X 46.582,Y -13.308,Z -39.863,A -90.000,B 90.000,C 0.000} C_DIS
LIN {X 47.104,Y -13.308,Z -40.044,A -90.000,B 90.000,C 0.000} C_DIS
LIN {X 47.653,Y -13.308,Z -40.227,A -90.000,B 90.000,C 0.000} C_DIS
LIN {X 47.974,Y -13.308,Z -40.326,A -90.000,B 90.000,C 0.000} C_DIS
LIN {X 48.092,Y -13.308,Z -40.359,A -90.000,B 90.000,C 0.000} C_DIS
LIN {X 48.182,Y -13.308,Z -40.378,A -90.000,B 90.000,C 0.000} C_DIS
LIN {X 48.190,Y -13.308,Z -40.391,A -90.000,B 90.000,C 0.000} C_DIS
LIN {X 48.202,Y -13.308,Z -40.402,A -90.000,B 90.000,C 0.000} C_DIS
LIN {X 48.253,Y -13.308,Z -40.440,A -90.000,B 90.000,C 0.000} C_DIS
LIN {X 48.357,Y -13.308,Z -40.506,A -90.000,B 90.000,C 0.000} C_DIS
LIN {X 48.531,Y -13.308,Z -40.607,A -90.000,B 90.000,C 0.000} C_DIS
LIN {X 48.962,Y -13.308,Z -40.842,A -90.000,B 90.000,C 0.000} C_DIS
LIN {X 49.651,Y -13.308,Z -41.199,A -90.000,B 90.000,C 0.000} C_DIS
LIN {X 49.716,Y -13.308,Z -41.231,A -90.000,B 90.000,C 0.000} C_DIS
LIN {X 49.716,Y -60.000,Z -41.231,A -90.000,B 90.000,C 0.000} C_DIS
LIN {X 60.190,Y -60.000,Z -48.340,A -90.000,B 90.000,C 0.000} C_DIS
LIN {X 60.190,Y -13.308,Z -48.340,A -90.000,B 90.000,C 0.000} C_DIS
LIN {X 61.516,Y -13.313,Z -49.182,A -90.000,B 90.000,C 0.000} C_DIS
LIN {X 61.701,Y -13.314,Z -49.302,A -90.000,B 90.000,C 0.000} C_DIS
LIN {X 61.839,Y -13.315,Z -49.386,A -90.000,B 90.000,C 0.000} C_DIS
LIN {X 63.708,Y -13.330,Z -50.439,A -90.000,B 90.000,C 0.000} C_DIS
LIN {X 64.045,Y -13.331,Z -50.628,A -90.000,B 90.000,C 0.000} C_DIS
LIN {X 65.079,Y -13.340,Z -51.169,A -90.000,B 90.000,C 0.000} C_DIS
LIN {X 65.705,Y -13.346,Z -51.492,A -90.000,B 90.000,C 0.000} C_DIS
LIN {X 66.268,Y -13.348,Z -51.789,A -90.000,B 90.000,C 0.000} C_DIS
LIN {X 68.316,Y -13.351,Z -52.888,A -90.000,B 90.000,C 0.000} C_DIS
LIN {X 69.255,Y -13.350,Z -53.424,A -90.000,B 90.000,C 0.000} C_DIS
LIN {X 70.524,Y -13.350,Z -54.145,A -90.000,B 90.000,C 0.000} C_DIS
LIN {X 72.538,Y -13.347,Z -55.372,A -90.000,B 90.000,C 0.000} C_DIS
LIN {X 72.703,Y -13.348,Z -55.472,A -90.000,B 90.000,C 0.000} C_DIS
LIN {X 74.844,Y -13.349,Z -56.875,A -90.000,B 90.000,C 0.000} C_DIS
LIN {X 75.168,Y -13.351,Z -57.091,A -90.000,B 90.000,C 0.000} C_DIS
LIN {X 75.564,Y -13.353,Z -57.373,A -90.000,B 90.000,C 0.000} C_DIS
LIN {X 76.884,Y -13.359,Z -58.327,A -90.000,B 90.000,C 0.000} C_DIS
LIN {X 76.965,Y -13.361,Z -58.385,A -90.000,B 90.000,C 0.000} C_DIS
LIN {X 77.398,Y -13.365,Z -58.723,A -90.000,B 90.000,C 0.000} C_DIS
LIN {X 78.444,Y -13.370,Z -59.566,A -90.000,B 90.000,C 0.000} C_DIS
LIN {X 78.444,Y -60.000,Z -59.566,A -90.000,B 90.000,C 0.000} C_DIS
LIN {X -120.015,Y -60.000,Z -242.845,A -90.000,B 90.000,C 0.000} C_DIS
LIN {X -120.015,Y -13.308,Z -242.845,A -90.000,B 90.000,C 0.000} C_DIS
LIN {X -118.906,Y -13.308,Z -242.083,A -90.000,B 90.000,C 0.000} C_DIS
LIN {X -116.192,Y -13.308,Z -240.198,A -90.000,B 90.000,C 0.000} C_DIS
LIN {X -111.781,Y -13.308,Z -237.182,A -90.000,B 90.000,C 0.000} C_DIS
LIN {X -108.836,Y -13.308,Z -235.172,A -90.000,B 90.000,C 0.000} C_DIS
LIN {X -101.187,Y -13.308,Z -230.020,A -90.000,B 90.000,C 0.000} C_DIS
LIN {X -96.536,Y -13.308,Z -226.939,A -90.000,B 90.000,C 0.000} C_DIS
LIN {X -93.299,Y -13.308,Z -224.812,A -90.000,B 90.000,C 0.000} C_DIS
LIN {X -88.178,Y -13.308,Z -221.506,A -90.000,B 90.000,C 0.000} C_DIS
LIN {X -85.188,Y -13.308,Z -219.598,A -90.000,B 90.000,C 0.000} C_DIS
LIN {X -78.759,Y -13.308,Z -215.582,A -90.000,B 90.000,C 0.000} C_DIS
LIN {X -76.843,Y -13.308,Z -214.390,A -90.000,B 90.000,C 0.000} C_DIS
LIN {X -71.994,Y -13.308,Z -211.390,A -90.000,B 90.000,C 0.000} C_DIS
LIN {X -68.387,Y -13.308,Z -209.172,A -90.000,B 90.000,C 0.000} C_DIS
LIN {X -63.893,Y -13.308,Z -206.389,A -90.000,B 90.000,C 0.000} C_DIS
LIN {X -60.700,Y -13.308,Z -204.430,A -90.000,B 90.000,C 0.000} C_DIS
LIN {X -57.876,Y -13.308,Z -202.654,A -90.000,B 90.000,C 0.000} C_DIS
LIN {X -53.918,Y -13.308,Z -200.196,A -90.000,B 90.000,C 0.000} C_DIS
LIN {X -49.553,Y -13.308,Z -197.383,A -90.000,B 90.000,C 0.000} C_DIS
LIN {X -48.583,Y -13.308,Z -196.751,A -90.000,B 90.000,C 0.000} C_DIS
LIN {X -44.130,Y -13.308,Z -193.765,A -90.000,B 90.000,C 0.000} C_DIS
LIN {X -43.893,Y -13.308,Z -193.604,A -90.000,B 90.000,C 0.000} C_DIS
LIN {X -41.159,Y -13.308,Z -191.691,A -90.000,B 90.000,C 0.000} C_DIS
LIN {X -39.923,Y -13.308,Z -190.830,A -90.000,B 90.000,C 0.000} C_DIS
LIN {X -36.511,Y -13.308,Z -188.354,A -90.000,B 90.000,C 0.000} C_DIS
LIN {X -33.359,Y -13.308,Z -186.004,A -90.000,B 90.000,C 0.000} C_DIS
LIN {X -32.971,Y -13.308,Z -185.698,A -90.000,B 90.000,C 0.000} C_DIS
LIN {X -30.500,Y -13.308,Z -183.780,A -90.000,B 90.000,C 0.000} C_DIS
LIN {X -30.012,Y -13.308,Z -183.373,A -90.000,B 90.000,C 0.000} C_DIS
LIN {X -27.791,Y -13.308,Z -181.551,A -90.000,B 90.000,C 0.000} C_DIS
LIN {X -27.270,Y -13.308,Z -181.086,A -90.000,B 90.000,C 0.000} C_DIS
LIN {X -25.588,Y -13.308,Z -179.604,A -90.000,B 90.000,C 0.000} C_DIS
LIN {X -23.905,Y -13.308,Z -177.984,A -90.000,B 90.000,C 0.000} C_DIS
LIN {X -23.344,Y -13.308,Z -177.441,A -90.000,B 90.000,C 0.000} C_DIS
LIN {X -21.450,Y -13.308,Z -175.418,A -90.000,B 90.000,C 0.000} C_DIS
LIN {X -20.165,Y -13.308,Z -173.869,A -90.000,B 90.000,C 0.000} C_DIS
LIN {X -19.676,Y -13.308,Z -173.286,A -90.000,B 90.000,C 0.000} C_DIS
LIN {X -18.316,Y -13.308,Z -171.411,A -90.000,B 90.000,C 0.000} C_DIS
LIN {X -18.076,Y -13.308,Z -171.084,A -90.000,B 90.000,C 0.000} C_DIS
LIN {X -16.700,Y -13.308,Z -168.896,A -90.000,B 90.000,C 0.000} C_DIS
LIN {X -16.331,Y -13.308,Z -168.199,A -90.000,B 90.000,C 0.000} C_DIS
LIN {X -15.442,Y -13.308,Z -166.538,A -90.000,B 90.000,C 0.000} C_DIS
LIN {X -15.122,Y -13.308,Z -165.762,A -90.000,B 90.000,C 0.000} C_DIS
LIN {X -14.559,Y -13.308,Z -164.453,A -90.000,B 90.000,C 0.000} C_DIS
LIN {X -14.350,Y -13.308,Z -163.654,A -90.000,B 90.000,C 0.000} C_DIS
LIN {X -14.134,Y -13.308,Z -162.919,A -90.000,B 90.000,C 0.000} C_DIS
LIN {X -14.122,Y -13.308,Z -162.520,A -90.000,B 90.000,C 0.000} C_DIS
LIN {X -14.084,Y -13.308,Z -162.065,A -90.000,B 90.000,C 0.000} C_DIS
LIN {X -14.127,Y -13.308,Z -161.860,A -90.000,B 90.000,C 0.000} C_DIS
LIN {X -14.181,Y -13.308,Z -161.523,A -90.000,B 90.000,C 0.000} C_DIS
LIN {X -14.236,Y -13.308,Z -161.399,A -90.000,B 90.000,C 0.000} C_DIS
LIN {X -14.325,Y -13.308,Z -161.180,A -90.000,B 90.000,C 0.000} C_DIS
LIN {X -14.402,Y -13.308,Z -160.987,A -90.000,B 90.000,C 0.000} C_DIS
LIN {X -14.630,Y -13.308,Z -160.616,A -90.000,B 90.000,C 0.000} C_DIS
LIN {X -14.928,Y -13.308,Z -160.093,A -90.000,B 90.000,C 0.000} C_DIS
LIN {X -15.069,Y -13.308,Z -159.902,A -90.000,B 90.000,C 0.000} C_DIS
LIN {X -15.602,Y -13.308,Z -159.038,A -90.000,B 90.000,C 0.000} C_DIS
LIN {X -15.940,Y -13.308,Z -158.609,A -90.000,B 90.000,C 0.000} C_DIS
LIN {X -16.495,Y -13.308,Z -157.837,A -90.000,B 90.000,C 0.000} C_DIS
LIN {X -16.773,Y -13.308,Z -157.540,A -90.000,B 90.000,C 0.000} C_DIS
LIN {X -17.789,Y -13.308,Z -156.328,A -90.000,B 90.000,C 0.000} C_DIS
LIN {X -18.335,Y -13.308,Z -155.793,A -90.000,B 90.000,C 0.000} C_DIS
LIN {X -19.651,Y -13.308,Z -154.405,A -90.000,B 90.000,C 0.000} C_DIS
LIN {X -20.129,Y -13.308,Z -153.966,A -90.000,B 90.000,C 0.000} C_DIS
LIN {X -20.727,Y -13.308,Z -153.406,A -90.000,B 90.000,C 0.000} C_DIS
LIN {X -22.371,Y -13.308,Z -151.820,A -90.000,B 90.000,C 0.000} C_DIS
LIN {X -23.558,Y -13.308,Z -150.696,A -90.000,B 90.000,C 0.000} C_DIS
LIN {X -25.502,Y -13.308,Z -148.786,A -90.000,B 90.000,C 0.000} C_DIS
LIN {X -26.713,Y -13.308,Z -147.527,A -90.000,B 90.000,C 0.000} C_DIS
LIN {X -28.735,Y -13.308,Z -145.363,A -90.000,B 90.000,C 0.000} C_DIS
LIN {X -29.061,Y -13.308,Z -145.007,A -90.000,B 90.000,C 0.000} C_DIS
LIN {X -30.261,Y -13.308,Z -143.545,A -90.000,B 90.000,C 0.000} C_DIS
LIN {X -32.098,Y -13.308,Z -141.257,A -90.000,B 90.000,C 0.000} C_DIS
LIN {X -32.385,Y -13.308,Z -140.869,A -90.000,B 90.000,C 0.000} C_DIS
LIN {X -33.785,Y -13.308,Z -138.639,A -90.000,B 90.000,C 0.000} C_DIS
LIN {X -34.971,Y -13.308,Z -136.781,A -90.000,B 90.000,C 0.000} C_DIS
LIN {X -35.003,Y -13.308,Z -136.730,A -90.000,B 90.000,C 0.000} C_DIS
LIN {X -35.170,Y -13.308,Z -136.440,A -90.000,B 90.000,C 0.000} C_DIS
LIN {X -36.140,Y -13.308,Z -134.571,A -90.000,B 90.000,C 0.000} C_DIS
LIN {X -37.317,Y -13.308,Z -132.318,A -90.000,B 90.000,C 0.000} C_DIS
LIN {X -38.978,Y -13.308,Z -128.623,A -90.000,B 90.000,C 0.000} C_DIS
LIN {X -39.120,Y -13.308,Z -128.300,A -90.000,B 90.000,C 0.000} C_DIS
LIN {X -39.415,Y -13.308,Z -127.586,A -90.000,B 90.000,C 0.000} C_DIS
LIN {X -40.412,Y -13.308,Z -125.153,A -90.000,B 90.000,C 0.000} C_DIS
LIN {X -41.049,Y -13.308,Z -123.624,A -90.000,B 90.000,C 0.000} C_DIS
LIN {X -41.371,Y -13.308,Z -122.839,A -90.000,B 90.000,C 0.000} C_DIS
LIN {X -42.027,Y -13.308,Z -121.415,A -90.000,B 90.000,C 0.000} C_DIS
LIN {X -42.286,Y -13.308,Z -120.967,A -90.000,B 90.000,C 0.000} C_DIS
LIN {X -42.773,Y -13.308,Z -120.114,A -90.000,B 90.000,C 0.000} C_DIS
LIN {X -43.309,Y -13.308,Z -119.360,A -90.000,B 90.000,C 0.000} C_DIS
LIN {X -43.831,Y -13.308,Z -118.615,A -90.000,B 90.000,C 0.000} C_DIS
LIN {X -44.436,Y -13.308,Z -117.851,A -90.000,B 90.000,C 0.000} C_DIS
LIN {X -45.460,Y -13.308,Z -116.579,A -90.000,B 90.000,C 0.000} C_DIS
LIN {X -46.004,Y -13.308,Z -115.920,A -90.000,B 90.000,C 0.000} C_DIS
LIN {X -47.698,Y -13.308,Z -113.894,A -90.000,B 90.000,C 0.000} C_DIS
LIN {X -49.223,Y -13.308,Z -112.063,A -90.000,B 90.000,C 0.000} C_DIS
LIN {X -50.027,Y -13.308,Z -111.092,A -90.000,B 90.000,C 0.000} C_DIS
LIN {X -52.532,Y -13.308,Z -107.954,A -90.000,B 90.000,C 0.000} C_DIS
LIN {X -55.159,Y -13.308,Z -104.431,A -90.000,B 90.000,C 0.000} C_DIS
LIN {X -55.266,Y -13.308,Z -104.287,A -90.000,B 90.000,C 0.000} C_DIS
LIN {X -55.945,Y -13.308,Z -103.354,A -90.000,B 90.000,C 0.000} C_DIS
LIN {X -57.718,Y -13.308,Z -100.911,A -90.000,B 90.000,C 0.000} C_DIS
LIN {X -59.764,Y -13.308,Z -98.100,A -90.000,B 90.000,C 0.000} C_DIS
LIN {X -60.816,Y -13.308,Z -96.732,A -90.000,B 90.000,C 0.000} C_DIS
LIN {X -61.854,Y -13.308,Z -95.363,A -90.000,B 90.000,C 0.000} C_DIS
LIN {X -62.390,Y -13.308,Z -94.740,A -90.000,B 90.000,C 0.000} C_DIS
LIN {X -63.692,Y -13.308,Z -93.172,A -90.000,B 90.000,C 0.000} C_DIS
LIN {X -64.382,Y -13.308,Z -92.461,A -90.000,B 90.000,C 0.000} C_DIS
LIN {X -65.570,Y -13.308,Z -91.176,A -90.000,B 90.000,C 0.000} C_DIS
LIN {X -65.979,Y -13.308,Z -90.798,A -90.000,B 90.000,C 0.000} C_DIS
LIN {X -66.353,Y -13.308,Z -90.450,A -90.000,B 90.000,C 0.000} C_DIS
LIN {X -67.346,Y -13.308,Z -89.496,A -90.000,B 90.000,C 0.000} C_DIS
LIN {X -67.756,Y -13.308,Z -89.163,A -90.000,B 90.000,C 0.000} C_DIS
LIN {X -68.113,Y -13.308,Z -88.862,A -90.000,B 90.000,C 0.000} C_DIS
LIN {X -69.173,Y -13.308,Z -87.960,A -90.000,B 90.000,C 0.000} C_DIS
LIN {X -71.063,Y -13.308,Z -86.519,A -90.000,B 90.000,C 0.000} C_DIS
LIN {X -71.306,Y -13.308,Z -86.339,A -90.000,B 90.000,C 0.000} C_DIS
LIN {X -72.593,Y -13.308,Z -85.436,A -90.000,B 90.000,C 0.000} C_DIS
LIN {X -73.222,Y -13.308,Z -85.005,A -90.000,B 90.000,C 0.000} C_DIS
LIN {X -74.516,Y -13.308,Z -84.158,A -90.000,B 90.000,C 0.000} C_DIS
LIN {X -75.281,Y -13.308,Z -83.664,A -90.000,B 90.000,C 0.000} C_DIS
LIN {X -76.474,Y -13.308,Z -82.929,A -90.000,B 90.000,C 0.000} C_DIS
LIN {X -77.277,Y -13.308,Z -82.431,A -90.000,B 90.000,C 0.000} C_DIS
LIN {X -78.190,Y -13.308,Z -81.879,A -90.000,B 90.000,C 0.000} C_DIS
LIN {X -79.010,Y -13.308,Z -81.395,A -90.000,B 90.000,C 0.000} C_DIS
LIN {X -79.835,Y -13.308,Z -80.890,A -90.000,B 90.000,C 0.000} C_DIS
LIN {X -80.586,Y -13.308,Z -80.450,A -90.000,B 90.000,C 0.000} C_DIS
LIN {X -81.335,Y -13.308,Z -79.964,A -90.000,B 90.000,C 0.000} C_DIS
LIN {X -81.874,Y -13.308,Z -79.633,A -90.000,B 90.000,C 0.000} C_DIS
LIN {X -82.261,Y -13.308,Z -79.372,A -90.000,B 90.000,C 0.000} C_DIS
LIN {X -83.164,Y -13.308,Z -78.722,A -90.000,B 90.000,C 0.000} C_DIS
LIN {X -83.421,Y -13.308,Z -78.546,A -90.000,B 90.000,C 0.000} C_DIS
LIN {X -84.300,Y -13.308,Z -77.851,A -90.000,B 90.000,C 0.000} C_DIS
LIN {X -84.806,Y -13.308,Z -77.434,A -90.000,B 90.000,C 0.000} C_DIS
LIN {X -85.251,Y -13.308,Z -77.053,A -90.000,B 90.000,C 0.000} C_DIS
LIN {X -86.185,Y -13.308,Z -76.240,A -90.000,B 90.000,C 0.000} C_DIS
LIN {X -86.645,Y -13.308,Z -75.842,A -90.000,B 90.000,C 0.000} C_DIS
LIN {X -87.187,Y -13.308,Z -75.401,A -90.000,B 90.000,C 0.000} C_DIS
LIN {X -87.641,Y -13.308,Z -75.092,A -90.000,B 90.000,C 0.000} C_DIS
LIN {X -87.797,Y -13.308,Z -74.980,A -90.000,B 90.000,C 0.000} C_DIS
LIN {X -88.575,Y -13.308,Z -74.522,A -90.000,B 90.000,C 0.000} C_DIS
LIN {X -89.178,Y -13.308,Z -74.211,A -90.000,B 90.000,C 0.000} C_DIS
LIN {X -90.091,Y -13.308,Z -73.796,A -90.000,B 90.000,C 0.000} C_DIS
LIN {X -90.576,Y -13.308,Z -73.600,A -90.000,B 90.000,C 0.000} C_DIS
LIN {X -91.094,Y -13.308,Z -73.419,A -90.000,B 90.000,C 0.000} C_DIS
LIN {X -91.203,Y -13.308,Z -73.379,A -90.000,B 90.000,C 0.000} C_DIS
LIN {X -91.614,Y -13.308,Z -73.253,A -90.000,B 90.000,C 0.000} C_DIS
LIN {X -92.034,Y -13.308,Z -73.120,A -90.000,B 90.000,C 0.000} C_DIS
LIN {X -92.467,Y -13.308,Z -72.993,A -90.000,B 90.000,C 0.000} C_DIS
LIN {X -92.702,Y -13.308,Z -72.945,A -90.000,B 90.000,C 0.000} C_DIS
LIN {X -93.226,Y -13.308,Z -72.808,A -90.000,B 90.000,C 0.000} C_DIS
LIN {X -93.939,Y -13.308,Z -72.678,A -90.000,B 90.000,C 0.000} C_DIS
LIN {X -94.064,Y -13.308,Z -72.647,A -90.000,B 90.000,C 0.000} C_DIS
LIN {X -94.886,Y -13.308,Z -72.491,A -90.000,B 90.000,C 0.000} C_DIS
LIN {X -95.460,Y -13.308,Z -72.407,A -90.000,B 90.000,C 0.000} C_DIS
LIN {X -95.847,Y -13.308,Z -72.324,A -90.000,B 90.000,C 0.000} C_DIS
LIN {X -96.273,Y -13.308,Z -72.222,A -90.000,B 90.000,C 0.000} C_DIS
LIN {X -96.947,Y -13.308,Z -72.107,A -90.000,B 90.000,C 0.000} C_DIS
LIN {X -97.359,Y -13.308,Z -72.009,A -90.000,B 90.000,C 0.000} C_DIS
LIN {X -97.386,Y -13.308,Z -71.999,A -90.000,B 90.000,C 0.000} C_DIS
LIN {X -97.624,Y -13.308,Z -71.933,A -90.000,B 90.000,C 0.000} C_DIS
LIN {X -98.336,Y -13.308,Z -71.719,A -90.000,B 90.000,C 0.000} C_DIS
LIN {X -98.507,Y -13.308,Z -71.678,A -90.000,B 90.000,C 0.000} C_DIS
LIN {X -98.921,Y -13.308,Z -71.528,A -90.000,B 90.000,C 0.000} C_DIS
LIN {X -99.885,Y -13.308,Z -71.115,A -90.000,B 90.000,C 0.000} C_DIS
LIN {X -100.133,Y -13.308,Z -71.025,A -90.000,B 90.000,C 0.000} C_DIS
LIN {X -100.528,Y -13.308,Z -70.829,A -90.000,B 90.000,C 0.000} C_DIS
LIN {X -101.600,Y -13.308,Z -70.189,A -90.000,B 90.000,C 0.000} C_DIS
LIN {X -101.797,Y -13.308,Z -70.084,A -90.000,B 90.000,C 0.000} C_DIS
LIN {X -102.167,Y -13.308,Z -69.844,A -90.000,B 90.000,C 0.000} C_DIS
LIN {X -102.307,Y -13.308,Z -69.743,A -90.000,B 90.000,C 0.000} C_DIS
LIN {X -103.617,Y -13.308,Z -68.671,A -90.000,B 90.000,C 0.000} C_DIS
LIN {X -103.788,Y -13.308,Z -68.530,A -90.000,B 90.000,C 0.000} C_DIS
LIN {X -103.823,Y -13.308,Z -68.499,A -90.000,B 90.000,C 0.000} C_DIS
LIN {X -104.859,Y -13.308,Z -67.447,A -90.000,B 90.000,C 0.000} C_DIS
LIN {X -105.083,Y -13.308,Z -67.217,A -90.000,B 90.000,C 0.000} C_DIS
LIN {X -105.428,Y -13.308,Z -66.848,A -90.000,B 90.000,C 0.000} C_DIS
LIN {X -105.719,Y -13.308,Z -66.519,A -90.000,B 90.000,C 0.000} C_DIS
LIN {X -105.919,Y -13.308,Z -66.284,A -90.000,B 90.000,C 0.000} C_DIS
LIN {X -106.542,Y -13.308,Z -65.529,A -90.000,B 90.000,C 0.000} C_DIS
LIN {X -106.771,Y -13.308,Z -65.249,A -90.000,B 90.000,C 0.000} C_DIS
LIN {X -106.919,Y -13.308,Z -65.057,A -90.000,B 90.000,C 0.000} C_DIS
LIN {X -107.042,Y -13.308,Z -64.894,A -90.000,B 90.000,C 0.000} C_DIS
LIN {X -107.337,Y -13.308,Z -64.491,A -90.000,B 90.000,C 0.000} C_DIS
LIN {X -107.755,Y -13.308,Z -63.884,A -90.000,B 90.000,C 0.000} C_DIS
LIN {X -107.981,Y -13.308,Z -63.548,A -90.000,B 90.000,C 0.000} C_DIS
LIN {X -108.848,Y -13.308,Z -62.163,A -90.000,B 90.000,C 0.000} C_DIS
LIN {X -109.076,Y -13.308,Z -61.786,A -90.000,B 90.000,C 0.000} C_DIS
LIN {X -109.204,Y -13.308,Z -61.556,A -90.000,B 90.000,C 0.000} C_DIS
LIN {X -109.702,Y -13.308,Z -60.510,A -90.000,B 90.000,C 0.000} C_DIS
LIN {X -110.140,Y -13.308,Z -59.273,A -90.000,B 90.000,C 0.000} C_DIS
LIN {X -110.293,Y -13.308,Z -58.827,A -90.000,B 90.000,C 0.000} C_DIS
LIN {X -110.416,Y -13.308,Z -58.416,A -90.000,B 90.000,C 0.000} C_DIS
LIN {X -110.569,Y -13.308,Z -57.846,A -90.000,B 90.000,C 0.000} C_DIS
LIN {X -110.663,Y -13.308,Z -57.433,A -90.000,B 90.000,C 0.000} C_DIS
LIN {X -110.719,Y -13.308,Z -57.152,A -90.000,B 90.000,C 0.000} C_DIS
LIN {X -110.821,Y -13.308,Z -56.468,A -90.000,B 90.000,C 0.000} C_DIS
LIN {X -110.927,Y -13.308,Z -55.939,A -90.000,B 90.000,C 0.000} C_DIS
LIN {X -110.955,Y -13.308,Z -55.737,A -90.000,B 90.000,C 0.000} C_DIS
LIN {X -111.026,Y -13.308,Z -55.397,A -90.000,B 90.000,C 0.000} C_DIS
LIN {X -111.069,Y -13.308,Z -55.119,A -90.000,B 90.000,C 0.000} C_DIS
LIN {X -111.121,Y -13.308,Z -54.892,A -90.000,B 90.000,C 0.000} C_DIS
LIN {X -111.160,Y -13.308,Z -54.681,A -90.000,B 90.000,C 0.000} C_DIS
LIN {X -111.241,Y -13.308,Z -54.406,A -90.000,B 90.000,C 0.000} C_DIS
LIN {X -111.262,Y -13.308,Z -54.329,A -90.000,B 90.000,C 0.000} C_DIS
LIN {X -111.301,Y -13.308,Z -54.214,A -90.000,B 90.000,C 0.000} C_DIS
LIN {X -111.309,Y -13.308,Z -54.194,A -90.000,B 90.000,C 0.000} C_DIS
LIN {X -111.343,Y -13.308,Z -54.149,A -90.000,B 90.000,C 0.000} C_DIS
LIN {X -111.653,Y -13.308,Z -53.706,A -90.000,B 90.000,C 0.000} C_DIS
LIN {X -111.932,Y -13.308,Z -53.283,A -90.000,B 90.000,C 0.000} C_DIS
LIN {X -112.225,Y -13.308,Z -52.803,A -90.000,B 90.000,C 0.000} C_DIS
LIN {X -112.445,Y -13.308,Z -52.380,A -90.000,B 90.000,C 0.000} C_DIS
LIN {X -112.660,Y -13.308,Z -51.919,A -90.000,B 90.000,C 0.000} C_DIS
LIN {X -112.748,Y -13.308,Z -51.718,A -90.000,B 90.000,C 0.000} C_DIS
LIN {X -112.913,Y -13.308,Z -51.318,A -90.000,B 90.000,C 0.000} C_DIS
LIN {X -113.067,Y -13.308,Z -50.877,A -90.000,B 90.000,C 0.000} C_DIS
LIN {X -113.208,Y -13.308,Z -50.375,A -90.000,B 90.000,C 0.000} C_DIS
LIN {X -113.310,Y -13.308,Z -49.963,A -90.000,B 90.000,C 0.000} C_DIS
LIN {X -113.403,Y -13.308,Z -49.518,A -90.000,B 90.000,C 0.000} C_DIS
LIN {X -113.472,Y -13.308,Z -48.795,A -90.000,B 90.000,C 0.000} C_DIS
LIN {X -113.497,Y -13.308,Z -48.493,A -90.000,B 90.000,C 0.000} C_DIS
LIN {X -113.510,Y -13.308,Z -48.301,A -90.000,B 90.000,C 0.000} C_DIS
LIN {X -113.499,Y -13.308,Z -47.861,A -90.000,B 90.000,C 0.000} C_DIS
LIN {X -113.486,Y -13.308,Z -47.733,A -90.000,B 90.000,C 0.000} C_DIS
LIN {X -113.364,Y -13.308,Z -46.806,A -90.000,B 90.000,C 0.000} C_DIS
LIN {X -113.158,Y -13.308,Z -46.006,A -90.000,B 90.000,C 0.000} C_DIS
LIN {X -112.864,Y -13.308,Z -45.245,A -90.000,B 90.000,C 0.000} C_DIS
LIN {X -112.753,Y -13.308,Z -45.008,A -90.000,B 90.000,C 0.000} C_DIS
LIN {X -112.673,Y -13.308,Z -44.850,A -90.000,B 90.000,C 0.000} C_DIS
LIN {X -112.820,Y -13.308,Z -44.550,A -90.000,B 90.000,C 0.000} C_DIS
LIN {X -113.126,Y -13.308,Z -43.902,A -90.000,B 90.000,C 0.000} C_DIS
LIN {X -113.309,Y -13.308,Z -43.507,A -90.000,B 90.000,C 0.000} C_DIS
LIN {X -113.363,Y -13.308,Z -43.382,A -90.000,B 90.000,C 0.000} C_DIS
LIN {X -113.585,Y -13.308,Z -42.824,A -90.000,B 90.000,C 0.000} C_DIS
LIN {X -113.914,Y -13.308,Z -41.889,A -90.000,B 90.000,C 0.000} C_DIS
LIN {X -114.087,Y -13.308,Z -41.313,A -90.000,B 90.000,C 0.000} C_DIS
LIN {X -114.178,Y -13.308,Z -40.956,A -90.000,B 90.000,C 0.000} C_DIS
LIN {X -114.269,Y -13.308,Z -40.557,A -90.000,B 90.000,C 0.000} C_DIS
LIN {X -114.363,Y -13.308,Z -40.112,A -90.000,B 90.000,C 0.000} C_DIS
LIN {X -114.426,Y -13.308,Z -39.739,A -90.000,B 90.000,C 0.000} C_DIS
LIN {X -114.473,Y -13.308,Z -39.279,A -90.000,B 90.000,C 0.000} C_DIS
LIN {X -114.510,Y -13.308,Z -38.880,A -90.000,B 90.000,C 0.000} C_DIS
LIN {X -114.520,Y -13.308,Z -38.758,A -90.000,B 90.000,C 0.000} C_DIS
LIN {X -114.524,Y -13.308,Z -38.491,A -90.000,B 90.000,C 0.000} C_DIS
LIN {X -114.516,Y -13.308,Z -38.041,A -90.000,B 90.000,C 0.000} C_DIS
LIN {X -114.511,Y -13.308,Z -37.847,A -90.000,B 90.000,C 0.000} C_DIS
LIN {X -114.488,Y -13.308,Z -37.550,A -90.000,B 90.000,C 0.000} C_DIS
LIN {X -114.450,Y -13.308,Z -37.276,A -90.000,B 90.000,C 0.000} C_DIS
LIN {X -114.428,Y -13.308,Z -37.113,A -90.000,B 90.000,C 0.000} C_DIS
LIN {X -114.382,Y -13.308,Z -36.830,A -90.000,B 90.000,C 0.000} C_DIS
LIN {X -114.316,Y -13.308,Z -36.557,A -90.000,B 90.000,C 0.000} C_DIS
LIN {X -114.207,Y -13.308,Z -36.130,A -90.000,B 90.000,C 0.000} C_DIS
LIN {X -114.067,Y -13.308,Z -35.687,A -90.000,B 90.000,C 0.000} C_DIS
LIN {X -113.971,Y -13.308,Z -35.423,A -90.000,B 90.000,C 0.000} C_DIS
LIN {X -113.819,Y -13.308,Z -35.030,A -90.000,B 90.000,C 0.000} C_DIS
LIN {X -113.700,Y -13.308,Z -34.765,A -90.000,B 90.000,C 0.000} C_DIS
LIN {X -113.504,Y -13.308,Z -34.392,A -90.000,B 90.000,C 0.000} C_DIS
LIN {X -113.361,Y -13.308,Z -34.139,A -90.000,B 90.000,C 0.000} C_DIS
LIN {X -113.120,Y -13.308,Z -33.790,A -90.000,B 90.000,C 0.000} C_DIS
LIN {X -112.945,Y -13.308,Z -33.547,A -90.000,B 90.000,C 0.000} C_DIS
LIN {X -112.658,Y -13.308,Z -33.221,A -90.000,B 90.000,C 0.000} C_DIS
LIN {X -112.445,Y -13.308,Z -32.992,A -90.000,B 90.000,C 0.000} C_DIS
LIN {X -111.954,Y -13.308,Z -32.518,A -90.000,B 90.000,C 0.000} C_DIS
LIN {X -111.892,Y -13.308,Z -32.453,A -90.000,B 90.000,C 0.000} C_DIS
LIN {X -111.706,Y -13.308,Z -32.216,A -90.000,B 90.000,C 0.000} C_DIS
LIN {X -111.148,Y -13.308,Z -31.458,A -90.000,B 90.000,C 0.000} C_DIS
LIN {X -110.817,Y -13.308,Z -31.042,A -90.000,B 90.000,C 0.000} C_DIS
LIN {X -110.543,Y -13.308,Z -30.730,A -90.000,B 90.000,C 0.000} C_DIS
LIN {X -110.184,Y -13.308,Z -30.333,A -90.000,B 90.000,C 0.000} C_DIS
LIN {X -109.796,Y -13.308,Z -29.942,A -90.000,B 90.000,C 0.000} C_DIS
LIN {X -109.382,Y -13.308,Z -29.559,A -90.000,B 90.000,C 0.000} C_DIS
LIN {X -108.978,Y -13.308,Z -29.202,A -90.000,B 90.000,C 0.000} C_DIS
LIN {X -108.645,Y -13.308,Z -28.912,A -90.000,B 90.000,C 0.000} C_DIS
LIN {X -108.201,Y -13.308,Z -28.541,A -90.000,B 90.000,C 0.000} C_DIS
LIN {X -107.679,Y -13.308,Z -28.169,A -90.000,B 90.000,C 0.000} C_DIS
LIN {X -107.360,Y -13.308,Z -27.951,A -90.000,B 90.000,C 0.000} C_DIS
LIN {X -106.738,Y -13.308,Z -27.599,A -90.000,B 90.000,C 0.000} C_DIS
LIN {X -106.356,Y -13.308,Z -27.395,A -90.000,B 90.000,C 0.000} C_DIS
LIN {X -105.596,Y -13.308,Z -27.061,A -90.000,B 90.000,C 0.000} C_DIS
LIN {X -105.203,Y -13.308,Z -26.905,A -90.000,B 90.000,C 0.000} C_DIS
LIN {X -104.249,Y -13.308,Z -26.592,A -90.000,B 90.000,C 0.000} C_DIS
LIN {X -103.230,Y -13.308,Z -26.297,A -90.000,B 90.000,C 0.000} C_DIS
LIN {X -102.855,Y -13.308,Z -26.182,A -90.000,B 90.000,C 0.000} C_DIS
LIN {X -102.318,Y -13.308,Z -26.022,A -90.000,B 90.000,C 0.000} C_DIS
LIN {X -102.188,Y -13.308,Z -25.837,A -90.000,B 90.000,C 0.000} C_DIS
LIN {X -101.987,Y -13.308,Z -25.560,A -90.000,B 90.000,C 0.000} C_DIS
LIN {X -101.875,Y -13.308,Z -25.415,A -90.000,B 90.000,C 0.000} C_DIS
LIN {X -101.722,Y -13.308,Z -25.175,A -90.000,B 90.000,C 0.000} C_DIS
LIN {X -101.496,Y -13.308,Z -24.854,A -90.000,B 90.000,C 0.000} C_DIS
LIN {X -101.443,Y -13.308,Z -24.779,A -90.000,B 90.000,C 0.000} C_DIS
LIN {X -101.349,Y -13.308,Z -24.658,A -90.000,B 90.000,C 0.000} C_DIS
LIN {X -101.221,Y -13.308,Z -24.454,A -90.000,B 90.000,C 0.000} C_DIS
LIN {X -101.011,Y -13.308,Z -24.168,A -90.000,B 90.000,C 0.000} C_DIS
LIN {X -100.708,Y -13.308,Z -23.784,A -90.000,B 90.000,C 0.000} C_DIS
LIN {X -100.613,Y -13.308,Z -23.663,A -90.000,B 90.000,C 0.000} C_DIS
LIN {X -100.328,Y -13.308,Z -23.327,A -90.000,B 90.000,C 0.000} C_DIS
LIN {X -100.123,Y -13.308,Z -23.125,A -90.000,B 90.000,C 0.000} C_DIS
LIN {X -99.793,Y -13.308,Z -22.816,A -90.000,B 90.000,C 0.000} C_DIS
LIN {X -99.581,Y -13.308,Z -22.649,A -90.000,B 90.000,C 0.000} C_DIS
LIN {X -99.237,Y -13.308,Z -22.408,A -90.000,B 90.000,C 0.000} C_DIS
LIN {X -98.989,Y -13.308,Z -22.257,A -90.000,B 90.000,C 0.000} C_DIS
LIN {X -98.616,Y -13.308,Z -22.056,A -90.000,B 90.000,C 0.000} C_DIS
LIN {X -98.223,Y -13.308,Z -21.900,A -90.000,B 90.000,C 0.000} C_DIS
LIN {X -97.528,Y -13.308,Z -21.716,A -90.000,B 90.000,C 0.000} C_DIS
LIN {X -97.109,Y -13.308,Z -21.657,A -90.000,B 90.000,C 0.000} C_DIS
LIN {X -96.366,Y -13.308,Z -21.641,A -90.000,B 90.000,C 0.000} C_DIS
LIN {X -96.052,Y -13.308,Z -21.671,A -90.000,B 90.000,C 0.000} C_DIS
LIN {X -95.977,Y -13.308,Z -21.481,A -90.000,B 90.000,C 0.000} C_DIS
LIN {X -95.890,Y -13.308,Z -21.287,A -90.000,B 90.000,C 0.000} C_DIS
LIN {X -95.827,Y -13.308,Z -21.173,A -90.000,B 90.000,C 0.000} C_DIS
LIN {X -95.571,Y -13.308,Z -20.627,A -90.000,B 90.000,C 0.000} C_DIS
LIN {X -95.535,Y -13.308,Z -20.556,A -90.000,B 90.000,C 0.000} C_DIS
LIN {X -95.330,Y -13.308,Z -20.237,A -90.000,B 90.000,C 0.000} C_DIS
LIN {X -95.067,Y -13.308,Z -19.848,A -90.000,B 90.000,C 0.000} C_DIS
LIN {X -94.900,Y -13.308,Z -19.652,A -90.000,B 90.000,C 0.000} C_DIS
LIN {X -94.633,Y -13.308,Z -19.349,A -90.000,B 90.000,C 0.000} C_DIS
LIN {X -94.431,Y -13.308,Z -19.158,A -90.000,B 90.000,C 0.000} C_DIS
LIN {X -94.125,Y -13.308,Z -18.886,A -90.000,B 90.000,C 0.000} C_DIS
LIN {X -93.355,Y -13.308,Z -18.349,A -90.000,B 90.000,C 0.000} C_DIS
LIN {X -93.270,Y -13.308,Z -18.297,A -90.000,B 90.000,C 0.000} C_DIS
LIN {X -92.897,Y -13.308,Z -18.096,A -90.000,B 90.000,C 0.000} C_DIS
LIN {X -92.548,Y -13.308,Z -17.938,A -90.000,B 90.000,C 0.000} C_DIS
LIN {X -91.932,Y -13.308,Z -17.681,A -90.000,B 90.000,C 0.000} C_DIS
LIN {X -91.799,Y -13.308,Z -17.630,A -90.000,B 90.000,C 0.000} C_DIS
LIN {X -91.723,Y -13.308,Z -17.604,A -90.000,B 90.000,C 0.000} C_DIS
LIN {X -91.667,Y -13.308,Z -17.588,A -90.000,B 90.000,C 0.000} C_DIS
LIN {X -90.801,Y -13.308,Z -17.337,A -90.000,B 90.000,C 0.000} C_DIS
LIN {X -90.553,Y -13.308,Z -17.271,A -90.000,B 90.000,C 0.000} C_DIS
LIN {X -90.120,Y -13.308,Z -17.189,A -90.000,B 90.000,C 0.000} C_DIS
LIN {X -89.756,Y -13.308,Z -17.140,A -90.000,B 90.000,C 0.000} C_DIS
LIN {X -89.085,Y -13.308,Z -17.059,A -90.000,B 90.000,C 0.000} C_DIS
LIN {X -88.660,Y -13.308,Z -17.027,A -90.000,B 90.000,C 0.000} C_DIS
LIN {X -87.543,Y -13.308,Z -17.066,A -90.000,B 90.000,C 0.000} C_DIS
LIN {X -87.142,Y -13.308,Z -17.082,A -90.000,B 90.000,C 0.000} C_DIS
LIN {X -87.101,Y -13.308,Z -17.085,A -90.000,B 90.000,C 0.000} C_DIS
LIN {X -86.705,Y -13.308,Z -17.147,A -90.000,B 90.000,C 0.000} C_DIS
LIN {X -86.399,Y -13.308,Z -17.211,A -90.000,B 90.000,C 0.000} C_DIS
LIN {X -86.268,Y -13.308,Z -17.011,A -90.000,B 90.000,C 0.000} C_DIS
LIN {X -86.116,Y -13.308,Z -16.794,A -90.000,B 90.000,C 0.000} C_DIS
LIN {X -86.078,Y -13.308,Z -16.744,A -90.000,B 90.000,C 0.000} C_DIS
LIN {X -85.836,Y -13.308,Z -16.440,A -90.000,B 90.000,C 0.000} C_DIS
LIN {X -85.794,Y -13.308,Z -16.391,A -90.000,B 90.000,C 0.000} C_DIS
LIN {X -85.521,Y -13.308,Z -16.115,A -90.000,B 90.000,C 0.000} C_DIS
LIN {X -85.465,Y -13.308,Z -16.063,A -90.000,B 90.000,C 0.000} C_DIS
LIN {X -85.111,Y -13.308,Z -15.777,A -90.000,B 90.000,C 0.000} C_DIS
LIN {X -84.790,Y -13.308,Z -15.534,A -90.000,B 90.000,C 0.000} C_DIS
LIN {X -84.406,Y -13.308,Z -15.289,A -90.000,B 90.000,C 0.000} C_DIS
LIN {X -84.187,Y -13.308,Z -15.172,A -90.000,B 90.000,C 0.000} C_DIS
LIN {X -83.705,Y -13.308,Z -14.934,A -90.000,B 90.000,C 0.000} C_DIS
LIN {X -83.553,Y -13.308,Z -14.865,A -90.000,B 90.000,C 0.000} C_DIS
LIN {X -83.046,Y -13.308,Z -14.664,A -90.000,B 90.000,C 0.000} C_DIS
LIN {X -82.516,Y -13.308,Z -14.499,A -90.000,B 90.000,C 0.000} C_DIS
LIN {X -82.209,Y -13.308,Z -14.415,A -90.000,B 90.000,C 0.000} C_DIS
LIN {X -82.010,Y -13.308,Z -14.356,A -90.000,B 90.000,C 0.000} C_DIS
LIN {X -81.497,Y -13.308,Z -14.256,A -90.000,B 90.000,C 0.000} C_DIS
LIN {X -80.997,Y -13.308,Z -14.158,A -90.000,B 90.000,C 0.000} C_DIS
LIN {X -80.790,Y -13.308,Z -14.123,A -90.000,B 90.000,C 0.000} C_DIS
LIN {X -80.131,Y -13.308,Z -14.054,A -90.000,B 90.000,C 0.000} C_DIS
LIN {X -79.838,Y -13.308,Z -14.021,A -90.000,B 90.000,C 0.000} C_DIS
LIN {X -79.351,Y -13.308,Z -13.978,A -90.000,B 90.000,C 0.000} C_DIS
LIN {X -78.855,Y -13.308,Z -13.965,A -90.000,B 90.000,C 0.000} C_DIS
LIN {X -78.488,Y -13.308,Z -13.960,A -90.000,B 90.000,C 0.000} C_DIS
LIN {X -78.215,Y -13.308,Z -13.963,A -90.000,B 90.000,C 0.000} C_DIS
LIN {X -77.748,Y -13.308,Z -13.972,A -90.000,B 90.000,C 0.000} C_DIS
LIN {X -77.278,Y -13.308,Z -14.009,A -90.000,B 90.000,C 0.000} C_DIS
LIN {X -76.768,Y -13.308,Z -14.073,A -90.000,B 90.000,C 0.000} C_DIS
LIN {X -76.024,Y -13.308,Z -14.189,A -90.000,B 90.000,C 0.000} C_DIS
LIN {X -75.497,Y -13.308,Z -14.294,A -90.000,B 90.000,C 0.000} C_DIS
LIN {X -75.037,Y -13.308,Z -14.416,A -90.000,B 90.000,C 0.000} C_DIS
LIN {X -74.451,Y -13.308,Z -14.585,A -90.000,B 90.000,C 0.000} C_DIS
LIN {X -73.163,Y -13.308,Z -15.019,A -90.000,B 90.000,C 0.000} C_DIS
LIN {X -72.577,Y -13.308,Z -15.243,A -90.000,B 90.000,C 0.000} C_DIS
LIN {X -72.343,Y -13.308,Z -15.337,A -90.000,B 90.000,C 0.000} C_DIS
LIN {X -70.993,Y -13.308,Z -15.975,A -90.000,B 90.000,C 0.000} C_DIS
LIN {X -70.560,Y -13.308,Z -16.189,A -90.000,B 90.000,C 0.000} C_DIS
LIN {X -70.199,Y -13.308,Z -16.372,A -90.000,B 90.000,C 0.000} C_DIS
LIN {X -68.409,Y -13.308,Z -17.302,A -90.000,B 90.000,C 0.000} C_DIS
LIN {X -67.422,Y -13.308,Z -17.821,A -90.000,B 90.000,C 0.000} C_DIS
LIN {X -67.154,Y -13.308,Z -17.966,A -90.000,B 90.000,C 0.000} C_DIS
LIN {X -66.307,Y -13.308,Z -18.406,A -90.000,B 90.000,C 0.000} C_DIS
LIN {X -65.746,Y -13.308,Z -18.719,A -90.000,B 90.000,C 0.000} C_DIS
LIN {X -65.262,Y -13.308,Z -18.959,A -90.000,B 90.000,C 0.000} C_DIS
LIN {X -64.480,Y -13.308,Z -19.397,A -90.000,B 90.000,C 0.000} C_DIS
LIN {X -63.900,Y -13.308,Z -19.677,A -90.000,B 90.000,C 0.000} C_DIS
LIN {X -63.397,Y -13.308,Z -19.961,A -90.000,B 90.000,C 0.000} C_DIS
LIN {X -62.960,Y -13.308,Z -20.164,A -90.000,B 90.000,C 0.000} C_DIS
LIN {X -62.373,Y -13.308,Z -20.482,A -90.000,B 90.000,C 0.000} C_DIS
LIN {X -61.663,Y -13.308,Z -20.809,A -90.000,B 90.000,C 0.000} C_DIS
LIN {X -61.328,Y -13.308,Z -20.989,A -90.000,B 90.000,C 0.000} C_DIS
LIN {X -60.640,Y -13.308,Z -21.311,A -90.000,B 90.000,C 0.000} C_DIS
LIN {X -60.517,Y -13.308,Z -21.369,A -90.000,B 90.000,C 0.000} C_DIS
LIN {X -59.533,Y -13.308,Z -21.802,A -90.000,B 90.000,C 0.000} C_DIS
LIN {X -59.147,Y -13.308,Z -21.945,A -90.000,B 90.000,C 0.000} C_DIS
LIN {X -58.490,Y -13.308,Z -22.207,A -90.000,B 90.000,C 0.000} C_DIS
LIN {X -58.095,Y -13.308,Z -22.328,A -90.000,B 90.000,C 0.000} C_DIS
LIN {X -57.149,Y -13.308,Z -22.651,A -90.000,B 90.000,C 0.000} C_DIS
LIN {X -55.585,Y -13.308,Z -23.072,A -90.000,B 90.000,C 0.000} C_DIS
LIN {X -54.917,Y -13.308,Z -23.237,A -90.000,B 90.000,C 0.000} C_DIS
LIN {X -53.353,Y -13.308,Z -23.557,A -90.000,B 90.000,C 0.000} C_DIS
LIN {X -53.008,Y -13.308,Z -23.620,A -90.000,B 90.000,C 0.000} C_DIS
LIN {X -51.889,Y -13.308,Z -23.848,A -90.000,B 90.000,C 0.000} C_DIS
LIN {X -51.179,Y -13.308,Z -23.974,A -90.000,B 90.000,C 0.000} C_DIS
LIN {X -50.347,Y -13.308,Z -24.127,A -90.000,B 90.000,C 0.000} C_DIS
LIN {X -49.177,Y -13.308,Z -24.338,A -90.000,B 90.000,C 0.000} C_DIS
LIN {X -48.310,Y -13.308,Z -24.502,A -90.000,B 90.000,C 0.000} C_DIS
LIN {X -47.051,Y -13.308,Z -24.749,A -90.000,B 90.000,C 0.000} C_DIS
LIN {X -45.198,Y -13.308,Z -25.143,A -90.000,B 90.000,C 0.000} C_DIS
LIN {X -43.673,Y -13.308,Z -25.474,A -90.000,B 90.000,C 0.000} C_DIS
LIN {X -42.525,Y -13.308,Z -25.740,A -90.000,B 90.000,C 0.000} C_DIS
LIN {X -41.755,Y -13.308,Z -25.912,A -90.000,B 90.000,C 0.000} C_DIS
LIN {X -41.007,Y -13.308,Z -26.091,A -90.000,B 90.000,C 0.000} C_DIS
LIN {X -39.851,Y -13.308,Z -26.360,A -90.000,B 90.000,C 0.000} C_DIS
LIN {X -38.535,Y -13.308,Z -26.687,A -90.000,B 90.000,C 0.000} C_DIS
LIN {X -37.619,Y -13.308,Z -26.904,A -90.000,B 90.000,C 0.000} C_DIS
LIN {X -37.202,Y -13.308,Z -27.002,A -90.000,B 90.000,C 0.000} C_DIS
LIN {X -37.147,Y -13.308,Z -27.014,A -90.000,B 90.000,C 0.000} C_DIS
LIN {X -35.981,Y -13.308,Z -27.029,A -90.000,B 90.000,C 0.000} C_DIS
LIN {X -35.725,Y -13.308,Z -27.042,A -90.000,B 90.000,C 0.000} C_DIS
LIN {X -35.397,Y -13.308,Z -27.049,A -90.000,B 90.000,C 0.000} C_DIS
LIN {X -33.619,Y -13.308,Z -27.066,A -90.000,B 90.000,C 0.000} C_DIS
LIN {X -32.617,Y -13.308,Z -27.137,A -90.000,B 90.000,C 0.000} C_DIS
LIN {X -32.046,Y -13.308,Z -27.171,A -90.000,B 90.000,C 0.000} C_DIS
LIN {X -31.696,Y -13.308,Z -27.198,A -90.000,B 90.000,C 0.000} C_DIS
LIN {X -29.698,Y -13.308,Z -27.426,A -90.000,B 90.000,C 0.000} C_DIS
LIN {X -27.459,Y -13.308,Z -27.682,A -90.000,B 90.000,C 0.000} C_DIS
LIN {X -25.368,Y -13.308,Z -27.961,A -90.000,B 90.000,C 0.000} C_DIS
LIN {X -25.128,Y -13.308,Z -27.990,A -90.000,B 90.000,C 0.000} C_DIS
LIN {X -22.658,Y -13.308,Z -28.382,A -90.000,B 90.000,C 0.000} C_DIS
LIN {X -22.179,Y -13.308,Z -28.460,A -90.000,B 90.000,C 0.000} C_DIS
LIN {X -20.346,Y -13.308,Z -28.808,A -90.000,B 90.000,C 0.000} C_DIS
LIN {X -19.641,Y -13.308,Z -28.947,A -90.000,B 90.000,C 0.000} C_DIS
LIN {X -17.897,Y -13.308,Z -29.298,A -90.000,B 90.000,C 0.000} C_DIS
LIN {X -16.263,Y -13.308,Z -29.642,A -90.000,B 90.000,C 0.000} C_DIS
LIN {X -15.248,Y -13.308,Z -29.845,A -90.000,B 90.000,C 0.000} C_DIS
LIN {X -14.521,Y -13.308,Z -30.003,A -90.000,B 90.000,C 0.000} C_DIS
LIN {X -13.060,Y -13.308,Z -30.286,A -90.000,B 90.000,C 0.000} C_DIS
LIN {X -12.317,Y -13.308,Z -30.433,A -90.000,B 90.000,C 0.000} C_DIS
LIN {X -10.772,Y -13.308,Z -30.734,A -90.000,B 90.000,C 0.000} C_DIS
LIN {X -9.414,Y -13.308,Z -31.029,A -90.000,B 90.000,C 0.000} C_DIS
LIN {X -9.023,Y -13.308,Z -31.106,A -90.000,B 90.000,C 0.000} C_DIS
LIN {X -6.457,Y -13.308,Z -31.641,A -90.000,B 90.000,C 0.000} C_DIS
LIN {X -5.049,Y -13.308,Z -31.896,A -90.000,B 90.000,C 0.000} C_DIS
LIN {X -3.487,Y -13.308,Z -32.201,A -90.000,B 90.000,C 0.000} C_DIS
LIN {X -2.573,Y -13.308,Z -32.367,A -90.000,B 90.000,C 0.000} C_DIS
LIN {X -0.602,Y -13.308,Z -32.675,A -90.000,B 90.000,C 0.000} C_DIS
LIN {X -0.236,Y -13.308,Z -32.738,A -90.000,B 90.000,C 0.000} C_DIS
LIN {X 1.454,Y -13.308,Z -32.988,A -90.000,B 90.000,C 0.000} C_DIS
LIN {X 2.262,Y -13.308,Z -33.125,A -90.000,B 90.000,C 0.000} C_DIS
LIN {X 4.512,Y -13.308,Z -33.523,A -90.000,B 90.000,C 0.000} C_DIS
LIN {X 5.019,Y -13.308,Z -33.615,A -90.000,B 90.000,C 0.000} C_DIS
LIN {X 5.126,Y -13.308,Z -33.633,A -90.000,B 90.000,C 0.000} C_DIS
LIN {X 7.096,Y -13.308,Z -34.028,A -90.000,B 90.000,C 0.000} C_DIS
LIN {X 7.489,Y -13.308,Z -34.098,A -90.000,B 90.000,C 0.000} C_DIS
LIN {X 7.682,Y -13.308,Z -34.136,A -90.000,B 90.000,C 0.000} C_DIS
LIN {X 8.931,Y -13.308,Z -34.416,A -90.000,B 90.000,C 0.000} C_DIS
LIN {X 10.289,Y -13.308,Z -34.735,A -90.000,B 90.000,C 0.000} C_DIS
LIN {X 11.481,Y -13.308,Z -35.023,A -90.000,B 90.000,C 0.000} C_DIS
LIN {X 12.513,Y -13.308,Z -35.279,A -90.000,B 90.000,C 0.000} C_DIS
LIN {X 14.305,Y -13.308,Z -35.693,A -90.000,B 90.000,C 0.000} C_DIS
LIN {X 15.384,Y -13.308,Z -35.888,A -90.000,B 90.000,C 0.000} C_DIS
LIN {X 16.015,Y -13.308,Z -35.994,A -90.000,B 90.000,C 0.000} C_DIS
LIN {X 16.698,Y -13.308,Z -36.045,A -90.000,B 90.000,C 0.000} C_DIS
LIN {X 17.419,Y -13.308,Z -36.066,A -90.000,B 90.000,C 0.000} C_DIS
LIN {X 17.825,Y -13.308,Z -36.063,A -90.000,B 90.000,C 0.000} C_DIS
LIN {X 18.606,Y -13.308,Z -36.000,A -90.000,B 90.000,C 0.000} C_DIS
LIN {X 18.697,Y -13.308,Z -35.995,A -90.000,B 90.000,C 0.000} C_DIS
LIN {X 20.076,Y -13.308,Z -35.844,A -90.000,B 90.000,C 0.000} C_DIS
LIN {X 20.407,Y -13.308,Z -35.810,A -90.000,B 90.000,C 0.000} C_DIS
LIN {X 21.039,Y -13.308,Z -35.750,A -90.000,B 90.000,C 0.000} C_DIS
LIN {X 21.115,Y -13.308,Z -35.739,A -90.000,B 90.000,C 0.000} C_DIS
LIN {X 21.204,Y -13.308,Z -35.731,A -90.000,B 90.000,C 0.000} C_DIS
LIN {X 22.402,Y -13.308,Z -35.662,A -90.000,B 90.000,C 0.000} C_DIS
LIN {X 22.812,Y -13.308,Z -35.647,A -90.000,B 90.000,C 0.000} C_DIS
LIN {X 23.725,Y -13.308,Z -35.635,A -90.000,B 90.000,C 0.000} C_DIS
LIN {X 23.903,Y -13.308,Z -35.635,A -90.000,B 90.000,C 0.000} C_DIS
LIN {X 24.526,Y -13.308,Z -35.650,A -90.000,B 90.000,C 0.000} C_DIS
LIN {X 24.967,Y -13.308,Z -35.668,A -90.000,B 90.000,C 0.000} C_DIS
LIN {X 25.541,Y -13.308,Z -35.696,A -90.000,B 90.000,C 0.000} C_DIS
LIN {X 26.455,Y -13.308,Z -35.756,A -90.000,B 90.000,C 0.000} C_DIS
LIN {X 26.817,Y -13.308,Z -35.785,A -90.000,B 90.000,C 0.000} C_DIS
LIN {X 27.236,Y -13.308,Z -35.823,A -90.000,B 90.000,C 0.000} C_DIS
LIN {X 27.663,Y -13.308,Z -35.870,A -90.000,B 90.000,C 0.000} C_DIS
LIN {X 29.094,Y -13.308,Z -36.010,A -90.000,B 90.000,C 0.000} C_DIS
LIN {X 29.689,Y -13.308,Z -36.081,A -90.000,B 90.000,C 0.000} C_DIS
LIN {X 30.662,Y -13.308,Z -36.182,A -90.000,B 90.000,C 0.000} C_DIS
LIN {X 32.965,Y -13.308,Z -36.470,A -90.000,B 90.000,C 0.000} C_DIS
LIN {X 33.123,Y -13.308,Z -36.494,A -90.000,B 90.000,C 0.000} C_DIS
LIN {X 34.090,Y -13.308,Z -36.623,A -90.000,B 90.000,C 0.000} C_DIS
LIN {X 34.560,Y -13.308,Z -36.696,A -90.000,B 90.000,C 0.000} C_DIS
LIN {X 35.239,Y -13.308,Z -36.814,A -90.000,B 90.000,C 0.000} C_DIS
LIN {X 35.657,Y -13.308,Z -36.877,A -90.000,B 90.000,C 0.000} C_DIS
LIN {X 36.133,Y -13.308,Z -36.960,A -90.000,B 90.000,C 0.000} C_DIS
LIN {X 37.658,Y -13.308,Z -37.250,A -90.000,B 90.000,C 0.000} C_DIS
LIN {X 38.139,Y -13.308,Z -37.348,A -90.000,B 90.000,C 0.000} C_DIS
LIN {X 38.465,Y -13.308,Z -37.434,A -90.000,B 90.000,C 0.000} C_DIS
LIN {X 39.118,Y -13.308,Z -37.588,A -90.000,B 90.000,C 0.000} C_DIS
LIN {X 40.816,Y -13.308,Z -38.002,A -90.000,B 90.000,C 0.000} C_DIS
LIN {X 41.284,Y -13.308,Z -38.141,A -90.000,B 90.000,C 0.000} C_DIS
LIN {X 41.842,Y -13.308,Z -38.319,A -90.000,B 90.000,C 0.000} C_DIS
LIN {X 43.487,Y -13.308,Z -38.797,A -90.000,B 90.000,C 0.000} C_DIS
LIN {X 43.897,Y -13.308,Z -38.920,A -90.000,B 90.000,C 0.000} C_DIS
LIN {X 46.609,Y -13.308,Z -39.873,A -90.000,B 90.000,C 0.000} C_DIS
LIN {X 47.102,Y -13.308,Z -40.078,A -90.000,B 90.000,C 0.000} C_DIS
LIN {X 49.502,Y -13.308,Z -41.123,A -90.000,B 90.000,C 0.000} C_DIS
LIN {X 49.774,Y -13.308,Z -41.262,A -90.000,B 90.000,C 0.000} C_DIS
LIN {X 52.087,Y -13.308,Z -42.490,A -90.000,B 90.000,C 0.000} C_DIS
LIN {X 52.579,Y -13.308,Z -42.757,A -90.000,B 90.000,C 0.000} C_DIS
LIN {X 52.705,Y -13.308,Z -42.827,A -90.000,B 90.000,C 0.000} C_DIS
LIN {X 55.120,Y -13.308,Z -44.350,A -90.000,B 90.000,C 0.000} C_DIS
LIN {X 55.508,Y -13.308,Z -44.614,A -90.000,B 90.000,C 0.000} C_DIS
LIN {X 57.720,Y -13.308,Z -46.256,A -90.000,B 90.000,C 0.000} C_DIS
LIN {X 60.139,Y -13.308,Z -48.299,A -90.000,B 90.000,C 0.000} C_DIS
LIN {X 60.190,Y -13.308,Z -48.340,A -90.000,B 90.000,C 0.000} C_DIS
LIN {X 61.265,Y -13.308,Z -49.022,A -90.000,B 90.000,C 0.000} C_DIS
LIN {X 61.702,Y -13.308,Z -49.302,A -90.000,B 90.000,C 0.000} C_DIS
LIN {X 61.822,Y -13.308,Z -49.376,A -90.000,B 90.000,C 0.000} C_DIS
LIN {X 64.018,Y -13.308,Z -50.609,A -90.000,B 90.000,C 0.000} C_DIS
LIN {X 65.060,Y -13.308,Z -51.152,A -90.000,B 90.000,C 0.000} C_DIS
LIN {X 65.717,Y -13.308,Z -51.489,A -90.000,B 90.000,C 0.000} C_DIS
LIN {X 66.145,Y -13.308,Z -51.714,A -90.000,B 90.000,C 0.000} C_DIS
LIN {X 68.330,Y -13.308,Z -52.885,A -90.000,B 90.000,C 0.000} C_DIS
LIN {X 69.031,Y -13.308,Z -53.287,A -90.000,B 90.000,C 0.000} C_DIS
LIN {X 70.534,Y -13.308,Z -54.141,A -90.000,B 90.000,C 0.000} C_DIS
LIN {X 72.711,Y -13.308,Z -55.467,A -90.000,B 90.000,C 0.000} C_DIS
LIN {X 74.775,Y -13.308,Z -56.819,A -90.000,B 90.000,C 0.000} C_DIS
LIN {X 75.177,Y -13.308,Z -57.086,A -90.000,B 90.000,C 0.000} C_DIS
LIN {X 75.514,Y -13.308,Z -57.324,A -90.000,B 90.000,C 0.000} C_DIS
LIN {X 76.976,Y -13.308,Z -58.378,A -90.000,B 90.000,C 0.000} C_DIS
LIN {X 77.483,Y -13.308,Z -58.772,A -90.000,B 90.000,C 0.000} C_DIS
LIN {X 78.470,Y -13.308,Z -59.565,A -90.000,B 90.000,C 0.000} C_DIS
LIN {X 78.763,Y -13.337,Z -59.800,A -90.000,B 90.000,C 0.000} C_DIS
LIN {X 79.027,Y -13.308,Z -60.009,A -90.000,B 90.000,C 0.000} C_DIS
LIN {X 79.263,Y -13.308,Z -60.194,A -90.000,B 90.000,C 0.000} C_DIS
LIN {X 79.265,Y -17.651,Z -60.195,A -90.000,B 90.000,C 0.000} C_DIS
LIN {X 79.277,Y -18.039,Z -60.205,A -90.000,B 90.000,C 0.000} C_DIS
LIN {X 79.291,Y -18.236,Z -60.215,A -90.000,B 90.000,C 0.000} C_DIS
LIN {X 79.318,Y -18.388,Z -60.236,A -90.000,B 90.000,C 0.000} C_DIS
LIN {X 79.372,Y -18.614,Z -60.277,A -90.000,B 90.000,C 0.000} C_DIS
LIN {X 79.474,Y -18.932,Z -60.355,A -90.000,B 90.000,C 0.000} C_DIS
LIN {X 79.570,Y -19.165,Z -60.426,A -90.000,B 90.000,C 0.000} C_DIS
LIN {X 79.660,Y -19.352,Z -60.491,A -90.000,B 90.000,C 0.000} C_DIS
LIN {X 79.745,Y -19.474,Z -60.551,A -90.000,B 90.000,C 0.000} C_DIS
LIN {X 79.898,Y -19.660,Z -60.652,A -90.000,B 90.000,C 0.000} C_DIS
LIN {X 80.007,Y -19.787,Z -60.718,A -90.000,B 90.000,C 0.000} C_DIS
LIN {X 80.009,Y -25.569,Z -60.719,A -90.000,B 90.000,C 0.000} C_DIS
LIN {X 80.015,Y -25.758,Z -60.722,A -90.000,B 90.000,C 0.000} C_DIS
LIN {X 80.030,Y -25.980,Z -60.731,A -90.000,B 90.000,C 0.000} C_DIS
LIN {X 80.089,Y -26.636,Z -60.762,A -90.000,B 90.000,C 0.000} C_DIS
LIN {X 80.144,Y -26.994,Z -60.787,A -90.000,B 90.000,C 0.000} C_DIS
LIN {X 80.195,Y -27.226,Z -60.807,A -90.000,B 90.000,C 0.000} C_DIS
LIN {X 80.219,Y -27.318,Z -60.815,A -90.000,B 90.000,C 0.000} C_DIS
LIN {X 80.263,Y -27.471,Z -60.826,A -90.000,B 90.000,C 0.000} C_DIS
LIN {X 80.304,Y -27.593,Z -60.833,A -90.000,B 90.000,C 0.000} C_DIS
LIN {X 80.342,Y -27.692,Z -60.833,A -90.000,B 90.000,C 0.000} C_DIS
LIN {X 80.376,Y -27.772,Z -60.829,A -90.000,B 90.000,C 0.000} C_DIS
LIN {X 80.407,Y -27.836,Z -60.819,A -90.000,B 90.000,C 0.000} C_DIS
LIN {X 80.435,Y -27.888,Z -60.805,A -90.000,B 90.000,C 0.000} C_DIS
LIN {X 80.461,Y -27.928,Z -60.785,A -90.000,B 90.000,C 0.000} C_DIS
LIN {X 80.473,Y -27.944,Z -60.773,A -90.000,B 90.000,C 0.000} C_DIS
LIN {X 80.494,Y -27.970,Z -60.745,A -90.000,B 90.000,C 0.000} C_DIS
LIN {X 80.514,Y -27.987,Z -60.712,A -90.000,B 90.000,C 0.000} C_DIS
LIN {X 80.532,Y -27.995,Z -60.675,A -90.000,B 90.000,C 0.000} C_DIS
LIN {X 80.548,Y -27.997,Z -60.632,A -90.000,B 90.000,C 0.000} C_DIS
LIN {X 80.562,Y -27.992,Z -60.585,A -90.000,B 90.000,C 0.000} C_DIS
LIN {X 80.575,Y -27.980,Z -60.533,A -90.000,B 90.000,C 0.000} C_DIS
LIN {X 80.587,Y -27.961,Z -60.476,A -90.000,B 90.000,C 0.000} C_DIS
LIN {X 80.598,Y -27.937,Z -60.415,A -90.000,B 90.000,C 0.000} C_DIS
LIN {X 80.618,Y -27.871,Z -60.277,A -90.000,B 90.000,C 0.000} C_DIS
LIN {X 80.636,Y -27.783,Z -60.122,A -90.000,B 90.000,C 0.000} C_DIS
LIN {X 80.655,Y -27.671,Z -59.949,A -90.000,B 90.000,C 0.000} C_DIS
LIN {X 80.675,Y -27.532,Z -59.759,A -90.000,B 90.000,C 0.000} C_DIS
LIN {X 80.700,Y -27.342,Z -59.551,A -90.000,B 90.000,C 0.000} C_DIS
LIN {X 80.729,Y -27.132,Z -59.327,A -90.000,B 90.000,C 0.000} C_DIS
LIN {X 80.766,Y -26.992,Z -59.087,A -90.000,B 90.000,C 0.000} C_DIS
LIN {X 80.810,Y -26.841,Z -58.831,A -90.000,B 90.000,C 0.000} C_DIS
LIN {X 80.865,Y -26.683,Z -58.560,A -90.000,B 90.000,C 0.000} C_DIS
LIN {X 80.932,Y -26.522,Z -58.274,A -90.000,B 90.000,C 0.000} C_DIS
LIN {X 80.970,Y -26.443,Z -58.125,A -90.000,B 90.000,C 0.000} C_DIS
LIN {X 81.012,Y -26.367,Z -57.973,A -90.000,B 90.000,C 0.000} C_DIS
LIN {X 81.058,Y -26.298,Z -57.817,A -90.000,B 90.000,C 0.000} C_DIS
LIN {X 81.107,Y -26.240,Z -57.658,A -90.000,B 90.000,C 0.000} C_DIS
LIN {X 81.161,Y -26.198,Z -57.496,A -90.000,B 90.000,C 0.000} C_DIS
LIN {X 81.219,Y -26.169,Z -57.330,A -90.000,B 90.000,C 0.000} C_DIS
LIN {X 81.282,Y -26.106,Z -57.160,A -90.000,B 90.000,C 0.000} C_DIS
LIN {X 81.349,Y -26.011,Z -56.988,A -90.000,B 90.000,C 0.000} C_DIS
LIN {X 81.422,Y -25.935,Z -56.812,A -90.000,B 90.000,C 0.000} C_DIS
LIN {X 81.499,Y -13.308,Z -56.633,A -90.000,B 90.000,C 0.000} C_DIS
LIN {X 81.700,Y -13.308,Z -56.182,A -90.000,B 90.000,C 0.000} C_DIS
LIN {X 82.134,Y -13.308,Z -55.110,A -90.000,B 90.000,C 0.000} C_DIS
LIN {X 82.335,Y -13.308,Z -54.666,A -90.000,B 90.000,C 0.000} C_DIS
LIN {X 83.331,Y -13.308,Z -52.811,A -90.000,B 90.000,C 0.000} C_DIS
LIN {X 83.577,Y -13.308,Z -52.389,A -90.000,B 90.000,C 0.000} C_DIS
LIN {X 84.737,Y -13.308,Z -50.685,A -90.000,B 90.000,C 0.000} C_DIS
LIN {X 85.025,Y -13.308,Z -50.291,A -90.000,B 90.000,C 0.000} C_DIS
LIN {X 86.337,Y -13.308,Z -48.714,A -90.000,B 90.000,C 0.000} C_DIS
LIN {X 86.664,Y -13.308,Z -48.352,A -90.000,B 90.000,C 0.000} C_DIS
LIN {X 88.117,Y -13.308,Z -46.880,A -90.000,B 90.000,C 0.000} C_DIS
LIN {X 88.479,Y -13.308,Z -46.553,A -90.000,B 90.000,C 0.000} C_DIS
LIN {X 90.061,Y -13.308,Z -45.164,A -90.000,B 90.000,C 0.000} C_DIS
LIN {X 91.716,Y -13.308,Z -43.876,A -90.000,B 90.000,C 0.000} C_DIS
LIN {X 92.110,Y -13.308,Z -43.588,A -90.000,B 90.000,C 0.000} C_DIS
LIN {X 93.780,Y -13.308,Z -42.419,A -90.000,B 90.000,C 0.000} C_DIS
LIN {X 95.417,Y -13.308,Z -41.383,A -90.000,B 90.000,C 0.000} C_DIS
LIN {X 95.838,Y -13.308,Z -41.136,A -90.000,B 90.000,C 0.000} C_DIS
LIN {X 97.376,Y -13.308,Z -40.260,A -90.000,B 90.000,C 0.000} C_DIS
LIN {X 98.805,Y -13.308,Z -39.523,A -90.000,B 90.000,C 0.000} C_DIS
LIN {X 98.814,Y -13.308,Z -39.518,A -90.000,B 90.000,C 0.000} C_DIS
LIN {X 98.814,Y -60.000,Z -39.518,A -90.000,B 90.000,C 0.000} C_DIS
LIN {X 99.842,Y -60.000,Z -87.116,A -90.000,B 90.000,C 0.000} C_DIS
LIN {X 99.842,Y -13.308,Z -87.116,A -90.000,B 90.000,C 0.000} C_DIS
LIN {X 99.870,Y -13.308,Z -87.476,A -90.000,B 90.000,C 0.000} C_DIS
LIN {X 99.925,Y -13.308,Z -88.260,A -90.000,B 90.000,C 0.000} C_DIS
LIN {X 100.078,Y -13.308,Z -88.517,A -90.000,B 90.000,C 0.000} C_DIS
LIN {X 100.820,Y -13.308,Z -89.872,A -90.000,B 90.000,C 0.000} C_DIS
LIN {X 100.968,Y -13.308,Z -90.148,A -90.000,B 90.000,C 0.000} C_DIS
LIN {X 101.529,Y -13.308,Z -91.330,A -90.000,B 90.000,C 0.000} C_DIS
LIN {X 101.700,Y -13.308,Z -91.755,A -90.000,B 90.000,C 0.000} C_DIS
LIN {X 101.785,Y -13.308,Z -91.973,A -90.000,B 90.000,C 0.000} C_DIS
LIN {X 102.135,Y -13.308,Z -92.892,A -90.000,B 90.000,C 0.000} C_DIS
LIN {X 102.180,Y -13.308,Z -93.034,A -90.000,B 90.000,C 0.000} C_DIS
LIN {X 102.478,Y -13.308,Z -94.013,A -90.000,B 90.000,C 0.000} C_DIS
LIN {X 102.601,Y -13.308,Z -94.452,A -90.000,B 90.000,C 0.000} C_DIS
LIN {X 102.875,Y -13.308,Z -95.543,A -90.000,B 90.000,C 0.000} C_DIS
LIN {X 103.113,Y -13.308,Z -96.595,A -90.000,B 90.000,C 0.000} C_DIS
LIN {X 103.399,Y -13.308,Z -97.927,A -90.000,B 90.000,C 0.000} C_DIS
LIN {X 103.671,Y -13.308,Z -99.255,A -90.000,B 90.000,C 0.000} C_DIS
LIN {X 103.967,Y -13.308,Z -100.795,A -90.000,B 90.000,C 0.000} C_DIS
LIN {X 104.297,Y -13.308,Z -102.630,A -90.000,B 90.000,C 0.000} C_DIS
LIN {X 104.349,Y -13.308,Z -102.941,A -90.000,B 90.000,C 0.000} C_DIS
LIN {X 104.546,Y -13.308,Z -104.112,A -90.000,B 90.000,C 0.000} C_DIS
LIN {X 104.771,Y -13.308,Z -105.486,A -90.000,B 90.000,C 0.000} C_DIS
LIN {X 104.891,Y -13.308,Z -106.239,A -90.000,B 90.000,C 0.000} C_DIS
LIN {X 105.141,Y -13.308,Z -107.882,A -90.000,B 90.000,C 0.000} C_DIS
LIN {X 105.239,Y -13.308,Z -108.547,A -90.000,B 90.000,C 0.000} C_DIS
LIN {X 105.508,Y -13.308,Z -110.483,A -90.000,B 90.000,C 0.000} C_DIS
LIN {X 105.705,Y -13.308,Z -111.966,A -90.000,B 90.000,C 0.000} C_DIS
LIN {X 105.859,Y -13.308,Z -113.211,A -90.000,B 90.000,C 0.000} C_DIS
LIN {X 105.999,Y -13.308,Z -114.402,A -90.000,B 90.000,C 0.000} C_DIS
LIN {X 106.204,Y -13.308,Z -116.355,A -90.000,B 90.000,C 0.000} C_DIS
LIN {X 106.252,Y -13.308,Z -116.824,A -90.000,B 90.000,C 0.000} C_DIS
LIN {X 106.456,Y -13.308,Z -119.127,A -90.000,B 90.000,C 0.000} C_DIS
LIN {X 106.637,Y -13.308,Z -121.538,A -90.000,B 90.000,C 0.000} C_DIS
LIN {X 106.794,Y -13.308,Z -123.736,A -90.000,B 90.000,C 0.000} C_DIS
LIN {X 106.841,Y -13.308,Z -124.542,A -90.000,B 90.000,C 0.000} C_DIS
LIN {X 106.973,Y -13.308,Z -126.674,A -90.000,B 90.000,C 0.000} C_DIS
LIN {X 106.993,Y -13.308,Z -127.015,A -90.000,B 90.000,C 0.000} C_DIS
LIN {X 107.021,Y -13.308,Z -127.642,A -90.000,B 90.000,C 0.000} C_DIS
LIN {X 107.118,Y -13.308,Z -129.571,A -90.000,B 90.000,C 0.000} C_DIS
LIN {X 107.143,Y -13.308,Z -130.385,A -90.000,B 90.000,C 0.000} C_DIS
LIN {X 107.208,Y -13.308,Z -132.255,A -90.000,B 90.000,C 0.000} C_DIS
LIN {X 107.221,Y -13.308,Z -133.226,A -90.000,B 90.000,C 0.000} C_DIS
LIN {X 107.257,Y -13.308,Z -135.164,A -90.000,B 90.000,C 0.000} C_DIS
LIN {X 107.263,Y -13.308,Z -137.284,A -90.000,B 90.000,C 0.000} C_DIS
LIN {X 107.259,Y -13.308,Z -138.312,A -90.000,B 90.000,C 0.000} C_DIS
LIN {X 107.224,Y -13.308,Z -140.740,A -90.000,B 90.000,C 0.000} C_DIS
LIN {X 107.216,Y -13.308,Z -141.106,A -90.000,B 90.000,C 0.000} C_DIS
LIN {X 107.204,Y -13.308,Z -141.948,A -90.000,B 90.000,C 0.000} C_DIS
LIN {X 107.081,Y -13.308,Z -145.626,A -90.000,B 90.000,C 0.000} C_DIS
LIN {X 107.062,Y -13.308,Z -145.984,A -90.000,B 90.000,C 0.000} C_DIS
LIN {X 106.869,Y -13.308,Z -149.436,A -90.000,B 90.000,C 0.000} C_DIS
LIN {X 106.552,Y -13.308,Z -153.317,A -90.000,B 90.000,C 0.000} C_DIS
LIN {X 106.516,Y -13.308,Z -153.739,A -90.000,B 90.000,C 0.000} C_DIS
LIN {X 106.120,Y -13.308,Z -157.660,A -90.000,B 90.000,C 0.000} C_DIS
LIN {X 105.676,Y -13.308,Z -161.554,A -90.000,B 90.000,C 0.000} C_DIS
LIN {X 105.210,Y -13.308,Z -165.369,A -90.000,B 90.000,C 0.000} C_DIS
LIN {X 104.772,Y -13.308,Z -168.875,A -90.000,B 90.000,C 0.000} C_DIS
LIN {X 104.664,Y -13.308,Z -169.687,A -90.000,B 90.000,C 0.000} C_DIS
LIN {X 104.328,Y -13.308,Z -172.302,A -90.000,B 90.000,C 0.000} C_DIS
LIN {X 104.185,Y -13.308,Z -173.331,A -90.000,B 90.000,C 0.000} C_DIS
LIN {X 103.893,Y -13.308,Z -175.511,A -90.000,B 90.000,C 0.000} C_DIS
LIN {X 103.720,Y -13.308,Z -176.702,A -90.000,B 90.000,C 0.000} C_DIS
LIN {X 103.456,Y -13.308,Z -178.570,A -90.000,B 90.000,C 0.000} C_DIS
LIN {X 103.248,Y -13.308,Z -179.959,A -90.000,B 90.000,C 0.000} C_DIS
LIN {X 102.995,Y -13.308,Z -181.601,A -90.000,B 90.000,C 0.000} C_DIS
LIN {X 102.621,Y -13.308,Z -183.964,A -90.000,B 90.000,C 0.000} C_DIS
LIN {X 101.931,Y -13.308,Z -188.253,A -90.000,B 90.000,C 0.000} C_DIS
LIN {X 101.669,Y -13.308,Z -189.905,A -90.000,B 90.000,C 0.000} C_DIS
LIN {X 101.459,Y -13.308,Z -191.263,A -90.000,B 90.000,C 0.000} C_DIS
LIN {X 101.427,Y -13.308,Z -191.466,A -90.000,B 90.000,C 0.000} C_DIS
LIN {X 101.280,Y -13.308,Z -192.383,A -90.000,B 90.000,C 0.000} C_DIS
LIN {X 101.054,Y -13.308,Z -193.844,A -90.000,B 90.000,C 0.000} C_DIS
LIN {X 100.841,Y -13.308,Z -195.132,A -90.000,B 90.000,C 0.000} C_DIS
LIN {X 100.574,Y -13.308,Z -196.807,A -90.000,B 90.000,C 0.000} C_DIS
LIN {X 100.309,Y -13.308,Z -198.341,A -90.000,B 90.000,C 0.000} C_DIS
LIN {X 99.974,Y -13.308,Z -200.358,A -90.000,B 90.000,C 0.000} C_DIS
LIN {X 99.688,Y -13.308,Z -201.949,A -90.000,B 90.000,C 0.000} C_DIS
LIN {X 99.502,Y -13.308,Z -203.021,A -90.000,B 90.000,C 0.000} C_DIS
LIN {X 99.213,Y -13.308,Z -204.709,A -90.000,B 90.000,C 0.000} C_DIS
LIN {X 98.413,Y -13.308,Z -209.053,A -90.000,B 90.000,C 0.000} C_DIS
LIN {X 98.284,Y -13.308,Z -209.749,A -90.000,B 90.000,C 0.000} C_DIS
LIN {X 98.226,Y -13.308,Z -210.052,A -90.000,B 90.000,C 0.000} C_DIS
LIN {X 97.149,Y -13.308,Z -215.443,A -90.000,B 90.000,C 0.000} C_DIS
LIN {X 95.937,Y -13.308,Z -220.956,A -90.000,B 90.000,C 0.000} C_DIS
LIN {X 95.361,Y -13.308,Z -223.287,A -90.000,B 90.000,C 0.000} C_DIS
LIN {X 94.565,Y -13.308,Z -226.526,A -90.000,B 90.000,C 0.000} C_DIS
LIN {X 93.841,Y -13.308,Z -229.169,A -90.000,B 90.000,C 0.000} C_DIS
LIN {X 93.011,Y -13.308,Z -232.213,A -90.000,B 90.000,C 0.000} C_DIS
LIN {X 92.090,Y -13.308,Z -235.280,A -90.000,B 90.000,C 0.000} C_DIS
LIN {X 91.217,Y -13.308,Z -238.205,A -90.000,B 90.000,C 0.000} C_DIS
LIN {X 91.108,Y -13.308,Z -238.556,A -90.000,B 90.000,C 0.000} C_DIS
LIN {X 90.022,Y -13.308,Z -241.906,A -90.000,B 90.000,C 0.000} C_DIS
LIN {X 89.490,Y -13.308,Z -243.561,A -90.000,B 90.000,C 0.000} C_DIS
LIN {X 89.490,Y -60.000,Z -243.561,A -90.000,B 90.000,C 0.000} C_DIS
LIN {X 101.240,Y -60.000,Z -88.584,A -90.000,B 90.000,C 0.000} C_DIS
LIN {X 101.240,Y -11.569,Z -88.584,A -90.000,B 90.000,C 0.000} C_DIS
LIN {X 101.276,Y -11.569,Z -88.649,A -90.000,B 90.000,C 0.000} C_DIS
LIN {X 101.829,Y -11.570,Z -89.660,A -90.000,B 90.000,C 0.000} C_DIS
LIN {X 101.962,Y -11.576,Z -89.912,A -90.000,B 90.000,C 0.000} C_DIS
LIN {X 102.433,Y -11.577,Z -90.901,A -90.000,B 90.000,C 0.000} C_DIS
LIN {X 102.529,Y -11.582,Z -91.109,A -90.000,B 90.000,C 0.000} C_DIS
LIN {X 102.699,Y -11.583,Z -91.532,A -90.000,B 90.000,C 0.000} C_DIS
LIN {X 103.088,Y -11.587,Z -92.529,A -90.000,B 90.000,C 0.000} C_DIS
LIN {X 103.139,Y -11.591,Z -92.667,A -90.000,B 90.000,C 0.000} C_DIS
LIN {X 103.483,Y -11.598,Z -93.764,A -90.000,B 90.000,C 0.000} C_DIS
LIN {X 103.590,Y -11.598,Z -94.142,A -90.000,B 90.000,C 0.000} C_DIS
LIN {X 103.888,Y -11.603,Z -95.290,A -90.000,B 90.000,C 0.000} C_DIS
LIN {X 104.157,Y -11.604,Z -96.477,A -90.000,B 90.000,C 0.000} C_DIS
LIN {X 104.418,Y -11.604,Z -97.693,A -90.000,B 90.000,C 0.000} C_DIS
LIN {X 104.694,Y -11.603,Z -99.044,A -90.000,B 90.000,C 0.000} C_DIS
LIN {X 104.996,Y -11.604,Z -100.600,A -90.000,B 90.000,C 0.000} C_DIS
LIN {X 105.252,Y -11.608,Z -101.996,A -90.000,B 90.000,C 0.000} C_DIS
LIN {X 105.361,Y -11.610,Z -102.585,A -90.000,B 90.000,C 0.000} C_DIS
LIN {X 105.712,Y -11.620,Z -104.595,A -90.000,B 90.000,C 0.000} C_DIS
LIN {X 105.958,Y -11.625,Z -106.068,A -90.000,B 90.000,C 0.000} C_DIS
LIN {X 106.305,Y -11.643,Z -108.187,A -90.000,B 90.000,C 0.000} C_DIS
LIN {X 106.682,Y -11.665,Z -110.669,A -90.000,B 90.000,C 0.000} C_DIS
LIN {X 106.844,Y -11.671,Z -111.825,A -90.000,B 90.000,C 0.000} C_DIS
LIN {X 106.998,Y -11.681,Z -112.945,A -90.000,B 90.000,C 0.000} C_DIS
LIN {X 107.162,Y -11.687,Z -114.264,A -90.000,B 90.000,C 0.000} C_DIS
LIN {X 107.342,Y -11.703,Z -115.769,A -90.000,B 90.000,C 0.000} C_DIS
LIN {X 107.438,Y -11.705,Z -116.681,A -90.000,B 90.000,C 0.000} C_DIS
LIN {X 107.627,Y -11.721,Z -118.556,A -90.000,B 90.000,C 0.000} C_DIS
LIN {X 107.670,Y -11.723,Z -119.019,A -90.000,B 90.000,C 0.000} C_DIS
LIN {X 107.869,Y -11.743,Z -121.304,A -90.000,B 90.000,C 0.000} C_DIS
LIN {X 108.049,Y -11.754,Z -123.647,A -90.000,B 90.000,C 0.000} C_DIS
LIN {X 108.072,Y -11.757,Z -123.969,A -90.000,B 90.000,C 0.000} C_DIS
LIN {X 108.212,Y -11.762,Z -126.148,A -90.000,B 90.000,C 0.000} C_DIS
LIN {X 108.255,Y -11.763,Z -126.841,A -90.000,B 90.000,C 0.000} C_DIS
LIN {X 108.389,Y -11.766,Z -129.502,A -90.000,B 90.000,C 0.000} C_DIS
LIN {X 108.399,Y -11.767,Z -129.788,A -90.000,B 90.000,C 0.000} C_DIS
LIN {X 108.482,Y -11.768,Z -132.201,A -90.000,B 90.000,C 0.000} C_DIS
LIN {X 108.495,Y -11.770,Z -132.901,A -90.000,B 90.000,C 0.000} C_DIS
LIN {X 108.534,Y -11.770,Z -135.066,A -90.000,B 90.000,C 0.000} C_DIS
LIN {X 108.541,Y -11.771,Z -137.248,A -90.000,B 90.000,C 0.000} C_DIS
LIN {X 108.543,Y -11.775,Z -138.232,A -90.000,B 90.000,C 0.000} C_DIS
LIN {X 108.513,Y -11.777,Z -140.583,A -90.000,B 90.000,C 0.000} C_DIS
LIN {X 108.498,Y -11.780,Z -141.647,A -90.000,B 90.000,C 0.000} C_DIS
LIN {X 108.492,Y -11.778,Z -141.968,A -90.000,B 90.000,C 0.000} C_DIS
LIN {X 108.385,Y -11.784,Z -145.356,A -90.000,B 90.000,C 0.000} C_DIS
LIN {X 108.372,Y -11.781,Z -145.669,A -90.000,B 90.000,C 0.000} C_DIS
LIN {X 108.262,Y -11.787,Z -147.783,A -90.000,B 90.000,C 0.000} C_DIS
LIN {X 108.190,Y -11.790,Z -149.117,A -90.000,B 90.000,C 0.000} C_DIS
LIN {X 108.165,Y -11.787,Z -149.509,A -90.000,B 90.000,C 0.000} C_DIS
LIN {X 108.022,Y -11.796,Z -151.392,A -90.000,B 90.000,C 0.000} C_DIS
LIN {X 107.896,Y -11.799,Z -152.974,A -90.000,B 90.000,C 0.000} C_DIS
LIN {X 107.823,Y -11.797,Z -153.828,A -90.000,B 90.000,C 0.000} C_DIS
LIN {X 107.658,Y -11.808,Z -155.587,A -90.000,B 90.000,C 0.000} C_DIS
LIN {X 107.482,Y -11.811,Z -157.373,A -90.000,B 90.000,C 0.000} C_DIS
LIN {X 107.442,Y -11.811,Z -157.765,A -90.000,B 90.000,C 0.000} C_DIS
LIN {X 107.284,Y -11.821,Z -159.247,A -90.000,B 90.000,C 0.000} C_DIS
LIN {X 107.031,Y -11.825,Z -161.520,A -90.000,B 90.000,C 0.000} C_DIS
LIN {X 106.878,Y -11.835,Z -162.857,A -90.000,B 90.000,C 0.000} C_DIS
LIN {X 106.642,Y -11.838,Z -164.826,A -90.000,B 90.000,C 0.000} C_DIS
LIN {X 106.369,Y -11.843,Z -167.077,A -90.000,B 90.000,C 0.000} C_DIS
LIN {X 106.267,Y -11.849,Z -167.941,A -90.000,B 90.000,C 0.000} C_DIS
LIN {X 106.177,Y -11.853,Z -168.694,A -90.000,B 90.000,C 0.000} C_DIS
LIN {X 106.036,Y -11.857,Z -169.811,A -90.000,B 90.000,C 0.000} C_DIS
LIN {X 105.775,Y -11.872,Z -171.957,A -90.000,B 90.000,C 0.000} C_DIS
LIN {X 105.713,Y -11.872,Z -172.441,A -90.000,B 90.000,C 0.000} C_DIS
LIN {X 105.586,Y -11.877,Z -173.394,A -90.000,B 90.000,C 0.000} C_DIS
LIN {X 105.343,Y -11.890,Z -175.311,A -90.000,B 90.000,C 0.000} C_DIS
LIN {X 105.296,Y -11.890,Z -175.656,A -90.000,B 90.000,C 0.000} C_DIS
LIN {X 105.155,Y -11.894,Z -176.662,A -90.000,B 90.000,C 0.000} C_DIS
LIN {X 104.916,Y -11.906,Z -178.432,A -90.000,B 90.000,C 0.000} C_DIS
LIN {X 104.723,Y -11.913,Z -179.782,A -90.000,B 90.000,C 0.000} C_DIS
LIN {X 104.470,Y -11.919,Z -181.477,A -90.000,B 90.000,C 0.000} C_DIS
LIN {X 104.261,Y -11.926,Z -182.850,A -90.000,B 90.000,C 0.000} C_DIS
LIN {X 103.863,Y -11.934,Z -185.384,A -90.000,B 90.000,C 0.000} C_DIS
LIN {X 103.527,Y -11.935,Z -187.481,A -90.000,B 90.000,C 0.000} C_DIS
LIN {X 103.089,Y -11.931,Z -190.210,A -90.000,B 90.000,C 0.000} C_DIS
LIN {X 102.858,Y -11.927,Z -191.670,A -90.000,B 90.000,C 0.000} C_DIS
LIN {X 102.706,Y -11.923,Z -192.603,A -90.000,B 90.000,C 0.000} C_DIS
LIN {X 102.488,Y -11.915,Z -193.968,A -90.000,B 90.000,C 0.000} C_DIS
LIN {X 102.445,Y -11.915,Z -194.228,A -90.000,B 90.000,C 0.000} C_DIS
LIN {X 102.257,Y -11.910,Z -195.334,A -90.000,B 90.000,C 0.000} C_DIS
LIN {X 101.988,Y -11.899,Z -196.956,A -90.000,B 90.000,C 0.000} C_DIS
LIN {X 101.955,Y -11.899,Z -197.147,A -90.000,B 90.000,C 0.000} C_DIS
LIN {X 101.723,Y -11.893,Z -198.459,A -90.000,B 90.000,C 0.000} C_DIS
LIN {X 101.363,Y -11.879,Z -200.532,A -90.000,B 90.000,C 0.000} C_DIS
LIN {X 101.075,Y -11.874,Z -202.108,A -90.000,B 90.000,C 0.000} C_DIS
LIN {X 100.581,Y -11.853,Z -204.854,A -90.000,B 90.000,C 0.000} C_DIS
LIN {X 100.531,Y -11.853,Z -205.124,A -90.000,B 90.000,C 0.000} C_DIS
LIN {X 99.644,Y -11.822,Z -209.766,A -90.000,B 90.000,C 0.000} C_DIS
LIN {X 99.549,Y -11.821,Z -210.249,A -90.000,B 90.000,C 0.000} C_DIS
LIN {X 98.446,Y -11.790,Z -215.594,A -90.000,B 90.000,C 0.000} C_DIS
LIN {X 98.187,Y -11.783,Z -216.744,A -90.000,B 90.000,C 0.000} C_DIS
LIN {X 97.161,Y -11.762,Z -221.290,A -90.000,B 90.000,C 0.000} C_DIS
LIN {X 95.806,Y -11.742,Z -226.690,A -90.000,B 90.000,C 0.000} C_DIS
LIN {X 95.722,Y -11.744,Z -227.017,A -90.000,B 90.000,C 0.000} C_DIS
LIN {X 95.480,Y -11.743,Z -227.899,A -90.000,B 90.000,C 0.000} C_DIS
LIN {X 94.199,Y -11.733,Z -232.537,A -90.000,B 90.000,C 0.000} C_DIS
LIN {X 94.138,Y -11.734,Z -232.752,A -90.000,B 90.000,C 0.000} C_DIS
LIN {X 93.584,Y -11.733,Z -234.590,A -90.000,B 90.000,C 0.000} C_DIS
LIN {X 92.601,Y -11.726,Z -237.849,A -90.000,B 90.000,C 0.000} C_DIS
LIN {X 92.353,Y -11.725,Z -238.668,A -90.000,B 90.000,C 0.000} C_DIS
LIN {X 92.304,Y -11.724,Z -238.821,A -90.000,B 90.000,C 0.000} C_DIS
LIN {X 91.623,Y -11.722,Z -240.920,A -90.000,B 90.000,C 0.000} C_DIS
LIN {X 90.762,Y -11.717,Z -243.561,A -90.000,B 90.000,C 0.000} C_DIS
LIN {X 90.762,Y -60.000,Z -243.561,A -90.000,B 90.000,C 0.000} C_DIS
LIN {X -120.015,Y -60.000,Z -241.274,A -90.000,B 90.000,C 0.000} C_DIS
LIN {X -120.015,Y -11.784,Z -241.274,A -90.000,B 90.000,C 0.000} C_DIS
LIN {X -116.908,Y -11.763,Z -239.150,A -90.000,B 90.000,C 0.000} C_DIS
LIN {X -111.000,Y -11.729,Z -235.164,A -90.000,B 90.000,C 0.000} C_DIS
LIN {X -109.515,Y -11.721,Z -234.163,A -90.000,B 90.000,C 0.000} C_DIS
LIN {X -101.999,Y -11.682,Z -229.164,A -90.000,B 90.000,C 0.000} C_DIS
LIN {X -96.866,Y -11.656,Z -225.807,A -90.000,B 90.000,C 0.000} C_DIS
LIN {X -94.065,Y -11.648,Z -223.980,A -90.000,B 90.000,C 0.000} C_DIS
LIN {X -88.763,Y -11.630,Z -220.589,A -90.000,B 90.000,C 0.000} C_DIS
LIN {X -85.763,Y -11.629,Z -218.677,A -90.000,B 90.000,C 0.000} C_DIS
LIN {X -80.447,Y -11.623,Z -215.366,A -90.000,B 90.000,C 0.000} C_DIS
LIN {X -77.383,Y -11.621,Z -213.460,A -90.000,B 90.000,C 0.000} C_DIS
LIN {X -74.476,Y -11.617,Z -211.670,A -90.000,B 90.000,C 0.000} C_DIS
LIN {X -72.238,Y -11.606,Z -210.307,A -90.000,B 90.000,C 0.000} C_DIS
LIN {X -68.162,Y -11.591,Z -207.827,A -90.000,B 90.000,C 0.000} C_DIS
LIN {X -66.724,Y -11.583,Z -206.953,A -90.000,B 90.000,C 0.000} C_DIS
LIN {X -64.409,Y -11.568,Z -205.549,A -90.000,B 90.000,C 0.000} C_DIS
LIN {X -62.531,Y -11.561,Z -204.412,A -90.000,B 90.000,C 0.000} C_DIS
LIN {X -61.477,Y -11.553,Z -203.781,A -90.000,B 90.000,C 0.000} C_DIS
LIN {X -60.626,Y -11.549,Z -203.259,A -90.000,B 90.000,C 0.000} C_DIS
LIN {X -58.422,Y -11.535,Z -201.906,A -90.000,B 90.000,C 0.000} C_DIS
LIN {X -56.656,Y -11.528,Z -200.824,A -90.000,B 90.000,C 0.000} C_DIS
LIN {X -54.566,Y -11.514,Z -199.558,A -90.000,B 90.000,C 0.000} C_DIS
LIN {X -54.405,Y -11.514,Z -199.458,A -90.000,B 90.000,C 0.000} C_DIS
LIN {X -52.200,Y -11.500,Z -198.072,A -90.000,B 90.000,C 0.000} C_DIS
LIN {X -49.926,Y -11.491,Z -196.630,A -90.000,B 90.000,C 0.000} C_DIS
LIN {X -48.865,Y -11.483,Z -195.955,A -90.000,B 90.000,C 0.000} C_DIS
LIN {X -46.282,Y -11.469,Z -194.262,A -90.000,B 90.000,C 0.000} C_DIS
LIN {X -44.334,Y -11.462,Z -192.973,A -90.000,B 90.000,C 0.000} C_DIS
LIN {X -44.083,Y -11.460,Z -192.804,A -90.000,B 90.000,C 0.000} C_DIS
LIN {X -42.246,Y -11.452,Z -191.543,A -90.000,B 90.000,C 0.000} C_DIS
LIN {X -40.350,Y -11.449,Z -190.229,A -90.000,B 90.000,C 0.000} C_DIS
LIN {X -38.837,Y -11.444,Z -189.147,A -90.000,B 90.000,C 0.000} C_DIS
LIN {X -36.930,Y -11.443,Z -187.768,A -90.000,B 90.000,C 0.000} C_DIS
LIN {X -35.223,Y -11.443,Z -186.495,A -90.000,B 90.000,C 0.000} C_DIS
LIN {X -33.729,Y -11.438,Z -185.394,A -90.000,B 90.000,C 0.000} C_DIS
LIN {X -32.128,Y -11.438,Z -184.147,A -90.000,B 90.000,C 0.000} C_DIS
LIN {X -30.940,Y -11.436,Z -183.233,A -90.000,B 90.000,C 0.000} C_DIS
LIN {X -30.826,Y -11.434,Z -183.145,A -90.000,B 90.000,C 0.000} C_DIS
LIN {X -29.261,Y -11.433,Z -181.856,A -90.000,B 90.000,C 0.000} C_DIS
LIN {X -28.444,Y -11.432,Z -181.190,A -90.000,B 90.000,C 0.000} C_DIS
LIN {X -28.247,Y -11.436,Z -181.017,A -90.000,B 90.000,C 0.000} C_DIS
LIN {X -26.993,Y -11.436,Z -179.906,A -90.000,B 90.000,C 0.000} C_DIS
LIN {X -26.004,Y -11.434,Z -179.037,A -90.000,B 90.000,C 0.000} C_DIS
LIN {X -23.975,Y -11.435,Z -177.078,A -90.000,B 90.000,C 0.000} C_DIS
LIN {X -23.850,Y -11.438,Z -176.944,A -90.000,B 90.000,C 0.000} C_DIS
LIN {X -23.373,Y -11.440,Z -176.428,A -90.000,B 90.000,C 0.000} C_DIS
LIN {X -22.074,Y -11.441,Z -175.036,A -90.000,B 90.000,C 0.000} C_DIS
LIN {X -21.994,Y -11.444,Z -174.939,A -90.000,B 90.000,C 0.000} C_DIS
LIN {X -21.395,Y -11.448,Z -174.201,A -90.000,B 90.000,C 0.000} C_DIS
LIN {X -20.471,Y -11.450,Z -173.083,A -90.000,B 90.000,C 0.000} C_DIS
LIN {X -20.280,Y -11.460,Z -172.815,A -90.000,B 90.000,C 0.000} C_DIS
LIN {X -19.961,Y -11.463,Z -172.363,A -90.000,B 90.000,C 0.000} C_DIS
LIN {X -18.968,Y -11.467,Z -170.983,A -90.000,B 90.000,C 0.000} C_DIS
LIN {X -18.746,Y -11.479,Z -170.631,A -90.000,B 90.000,C 0.000} C_DIS
LIN {X -18.048,Y -11.484,Z -169.500,A -90.000,B 90.000,C 0.000} C_DIS
LIN {X -17.595,Y -11.490,Z -168.754,A -90.000,B 90.000,C 0.000} C_DIS
LIN {X -17.437,Y -11.501,Z -168.461,A -90.000,B 90.000,C 0.000} C_DIS
LIN {X -16.650,Y -11.506,Z -166.958,A -90.000,B 90.000,C 0.000} C_DIS
LIN {X -16.385,Y -11.509,Z -166.451,A -90.000,B 90.000,C 0.000} C_DIS
LIN {X -16.254,Y -11.521,Z -166.154,A -90.000,B 90.000,C 0.000} C_DIS
LIN {X -15.969,Y -11.519,Z -165.474,A -90.000,B 90.000,C 0.000} C_DIS
LIN {X -15.533,Y -11.521,Z -164.447,A -90.000,B 90.000,C 0.000} C_DIS
LIN {X -15.440,Y -11.537,Z -164.151,A -90.000,B 90.000,C 0.000} C_DIS
LIN {X -15.226,Y -11.529,Z -163.397,A -90.000,B 90.000,C 0.000} C_DIS
LIN {X -15.073,Y -11.529,Z -162.874,A -90.000,B 90.000,C 0.000} C_DIS
LIN {X -15.060,Y -11.538,Z -162.772,A -90.000,B 90.000,C 0.000} C_DIS
LIN {X -15.035,Y -11.531,Z -162.444,A -90.000,B 90.000,C 0.000} C_DIS
LIN {X -15.007,Y -11.530,Z -162.122,A -90.000,B 90.000,C 0.000} C_DIS
LIN {X -15.005,Y -11.522,Z -162.057,A -90.000,B 90.000,C 0.000} C_DIS
LIN {X -15.048,Y -11.521,Z -161.778,A -90.000,B 90.000,C 0.000} C_DIS
LIN {X -15.093,Y -11.498,Z -161.547,A -90.000,B 90.000,C 0.000} C_DIS
LIN {X -15.163,Y -11.497,Z -161.369,A -90.000,B 90.000,C 0.000} C_DIS
LIN {X -15.215,Y -11.487,Z -161.241,A -90.000,B 90.000,C 0.000} C_DIS
LIN {X -15.313,Y -11.466,Z -160.987,A -90.000,B 90.000,C 0.000} C_DIS
LIN {X -15.535,Y -11.465,Z -160.592,A -90.000,B 90.000,C 0.000} C_DIS
LIN {X -15.588,Y -11.461,Z -160.488,A -90.000,B 90.000,C 0.000} C_DIS
LIN {X -15.695,Y -11.447,Z -160.281,A -90.000,B 90.000,C 0.000} C_DIS
LIN {X -15.778,Y -11.441,Z -160.116,A -90.000,B 90.000,C 0.000} C_DIS
LIN {X -16.193,Y -11.440,Z -159.438,A -90.000,B 90.000,C 0.000} C_DIS
LIN {X -16.218,Y -11.438,Z -159.400,A -90.000,B 90.000,C 0.000} C_DIS
LIN {X -16.374,Y -11.418,Z -159.115,A -90.000,B 90.000,C 0.000} C_DIS
LIN {X -16.551,Y -11.416,Z -158.868,A -90.000,B 90.000,C 0.000} C_DIS
LIN {X -16.841,Y -11.415,Z -158.462,A -90.000,B 90.000,C 0.000} C_DIS
LIN {X -16.992,Y -11.412,Z -158.236,A -90.000,B 90.000,C 0.000} C_DIS
LIN {X -17.084,Y -11.404,Z -158.101,A -90.000,B 90.000,C 0.000} C_DIS
LIN {X -17.185,Y -11.394,Z -157.946,A -90.000,B 90.000,C 0.000} C_DIS
LIN {X -17.819,Y -11.393,Z -157.188,A -90.000,B 90.000,C 0.000} C_DIS
LIN {X -18.049,Y -11.392,Z -156.907,A -90.000,B 90.000,C 0.000} C_DIS
LIN {X -18.213,Y -11.388,Z -156.693,A -90.000,B 90.000,C 0.000} C_DIS
LIN {X -18.344,Y -11.379,Z -156.524,A -90.000,B 90.000,C 0.000} C_DIS
LIN {X -18.706,Y -11.375,Z -156.145,A -90.000,B 90.000,C 0.000} C_DIS
LIN {X -19.563,Y -11.375,Z -155.240,A -90.000,B 90.000,C 0.000} C_DIS
LIN {X -19.876,Y -11.373,Z -154.899,A -90.000,B 90.000,C 0.000} C_DIS
LIN {X -20.000,Y -11.371,Z -154.759,A -90.000,B 90.000,C 0.000} C_DIS
LIN {X -20.087,Y -11.368,Z -154.662,A -90.000,B 90.000,C 0.000} C_DIS
LIN {X -21.047,Y -11.362,Z -153.737,A -90.000,B 90.000,C 0.000} C_DIS
LIN {X -21.993,Y -11.362,Z -152.823,A -90.000,B 90.000,C 0.000} C_DIS
LIN {X -22.721,Y -11.357,Z -152.090,A -90.000,B 90.000,C 0.000} C_DIS
LIN {X -23.844,Y -11.351,Z -150.988,A -90.000,B 90.000,C 0.000} C_DIS
LIN {X -24.916,Y -11.350,Z -149.934,A -90.000,B 90.000,C 0.000} C_DIS
LIN {X -25.787,Y -11.346,Z -149.048,A -90.000,B 90.000,C 0.000} C_DIS
LIN {X -26.978,Y -11.341,Z -147.774,A -90.000,B 90.000,C 0.000} C_DIS
LIN {X -28.175,Y -11.341,Z -146.493,A -90.000,B 90.000,C 0.000} C_DIS
LIN {X -28.676,Y -11.341,Z -145.952,A -90.000,B 90.000,C 0.000} C_DIS
LIN {X -29.076,Y -11.340,Z -145.511,A -90.000,B 90.000,C 0.000} C_DIS
LIN {X -29.314,Y -11.338,Z -145.239,A -90.000,B 90.000,C 0.000} C_DIS
LIN {X -29.423,Y -11.338,Z -145.107,A -90.000,B 90.000,C 0.000} C_DIS
LIN {X -29.660,Y -11.337,Z -144.811,A -90.000,B 90.000,C 0.000} C_DIS
LIN {X -30.515,Y -11.335,Z -143.749,A -90.000,B 90.000,C 0.000} C_DIS
LIN {X -32.113,Y -11.335,Z -141.759,A -90.000,B 90.000,C 0.000} C_DIS
LIN {X -32.421,Y -11.335,Z -141.367,A -90.000,B 90.000,C 0.000} C_DIS
LIN {X -32.699,Y -11.334,Z -140.968,A -90.000,B 90.000,C 0.000} C_DIS
LIN {X -32.946,Y -11.334,Z -140.571,A -90.000,B 90.000,C 0.000} C_DIS
LIN {X -35.244,Y -11.333,Z -136.929,A -90.000,B 90.000,C 0.000} C_DIS
LIN {X -35.479,Y -11.332,Z -136.503,A -90.000,B 90.000,C 0.000} C_DIS
LIN {X -36.504,Y -11.332,Z -134.538,A -90.000,B 90.000,C 0.000} C_DIS
LIN {X -37.574,Y -11.331,Z -132.477,A -90.000,B 90.000,C 0.000} C_DIS
LIN {X -39.275,Y -11.331,Z -128.691,A -90.000,B 90.000,C 0.000} C_DIS
LIN {X -39.398,Y -11.331,Z -128.411,A -90.000,B 90.000,C 0.000} C_DIS
LIN {X -40.852,Y -11.332,Z -124.897,A -90.000,B 90.000,C 0.000} C_DIS
LIN {X -41.662,Y -11.335,Z -122.980,A -90.000,B 90.000,C 0.000} C_DIS
LIN {X -41.941,Y -11.335,Z -122.381,A -90.000,B 90.000,C 0.000} C_DIS
LIN {X -42.353,Y -11.336,Z -121.508,A -90.000,B 90.000,C 0.000} C_DIS
LIN {X -43.052,Y -11.336,Z -120.292,A -90.000,B 90.000,C 0.000} C_DIS
LIN {X -43.076,Y -11.335,Z -120.251,A -90.000,B 90.000,C 0.000} C_DIS
LIN {X -43.995,Y -11.334,Z -118.942,A -90.000,B 90.000,C 0.000} C_DIS
LIN {X -44.089,Y -11.334,Z -118.807,A -90.000,B 90.000,C 0.000} C_DIS
LIN {X -44.317,Y -11.334,Z -118.516,A -90.000,B 90.000,C 0.000} C_DIS
LIN {X -45.813,Y -11.333,Z -116.638,A -90.000,B 90.000,C 0.000} C_DIS
LIN {X -47.786,Y -11.331,Z -114.256,A -90.000,B 90.000,C 0.000} C_DIS
LIN {X -49.693,Y -11.329,Z -111.946,A -90.000,B 90.000,C 0.000} C_DIS
LIN {X -50.187,Y -11.330,Z -111.354,A -90.000,B 90.000,C 0.000} C_DIS
LIN {X -51.808,Y -11.330,Z -109.331,A -90.000,B 90.000,C 0.000} C_DIS
LIN {X -52.644,Y -11.331,Z -108.292,A -90.000,B 90.000,C 0.000} C_DIS
LIN {X -55.091,Y -11.333,Z -105.045,A -90.000,B 90.000,C 0.000} C_DIS
LIN {X -57.441,Y -11.335,Z -101.848,A -90.000,B 90.000,C 0.000} C_DIS
LIN {X -59.597,Y -11.341,Z -98.937,A -90.000,B 90.000,C 0.000} C_DIS
LIN {X -60.130,Y -11.346,Z -98.261,A -90.000,B 90.000,C 0.000} C_DIS
LIN {X -61.414,Y -11.352,Z -96.630,A -90.000,B 90.000,C 0.000} C_DIS
LIN {X -61.817,Y -11.353,Z -96.106,A -90.000,B 90.000,C 0.000} C_DIS
LIN {X -62.216,Y -11.363,Z -95.655,A -90.000,B 90.000,C 0.000} C_DIS
LIN {X -62.712,Y -11.366,Z -95.098,A -90.000,B 90.000,C 0.000} C_DIS
LIN {X -63.131,Y -11.371,Z -94.626,A -90.000,B 90.000,C 0.000} C_DIS
LIN {X -63.750,Y -11.375,Z -93.904,A -90.000,B 90.000,C 0.000} C_DIS
LIN {X -64.016,Y -11.384,Z -93.638,A -90.000,B 90.000,C 0.000} C_DIS
LIN {X -64.107,Y -11.388,Z -93.546,A -90.000,B 90.000,C 0.000} C_DIS
LIN {X -64.807,Y -11.394,Z -92.853,A -90.000,B 90.000,C 0.000} C_DIS
LIN {X -65.214,Y -11.401,Z -92.447,A -90.000,B 90.000,C 0.000} C_DIS
LIN {X -65.623,Y -11.405,Z -92.022,A -90.000,B 90.000,C 0.000} C_DIS
LIN {X -66.040,Y -11.423,Z -91.650,A -90.000,B 90.000,C 0.000} C_DIS
LIN {X -66.662,Y -11.431,Z -91.103,A -90.000,B 90.000,C 0.000} C_DIS
LIN {X -67.491,Y -11.439,Z -90.341,A -90.000,B 90.000,C 0.000} C_DIS
LIN {X -67.845,Y -11.454,Z -90.057,A -90.000,B 90.000,C 0.000} C_DIS
LIN {X -68.367,Y -11.460,Z -89.646,A -90.000,B 90.000,C 0.000} C_DIS
LIN {X -68.844,Y -11.468,Z -89.268,A -90.000,B 90.000,C 0.000} C_DIS
LIN {X -69.441,Y -11.474,Z -88.779,A -90.000,B 90.000,C 0.000} C_DIS
LIN {X -69.684,Y -11.482,Z -88.595,A -90.000,B 90.000,C 0.000} C_DIS
LIN {X -70.288,Y -11.487,Z -88.148,A -90.000,B 90.000,C 0.000} C_DIS
LIN {X -71.659,Y -11.505,Z -87.154,A -90.000,B 90.000,C 0.000} C_DIS
LIN {X -71.815,Y -11.508,Z -87.045,A -90.000,B 90.000,C 0.000} C_DIS
LIN {X -72.650,Y -11.513,Z -86.472,A -90.000,B 90.000,C 0.000} C_DIS
LIN {X -73.485,Y -11.519,Z -85.907,A -90.000,B 90.000,C 0.000} C_DIS
LIN {X -73.754,Y -11.523,Z -85.731,A -90.000,B 90.000,C 0.000} C_DIS
LIN {X -74.777,Y -11.525,Z -85.070,A -90.000,B 90.000,C 0.000} C_DIS
LIN {X -75.607,Y -11.528,Z -84.537,A -90.000,B 90.000,C 0.000} C_DIS
LIN {X -75.988,Y -11.529,Z -84.299,A -90.000,B 90.000,C 0.000} C_DIS
LIN {X -77.746,Y -11.525,Z -83.205,A -90.000,B 90.000,C 0.000} C_DIS
LIN {X -78.786,Y -11.516,Z -82.558,A -90.000,B 90.000,C 0.000} C_DIS
LIN {X -79.195,Y -11.513,Z -82.309,A -90.000,B 90.000,C 0.000} C_DIS
LIN {X -79.492,Y -11.507,Z -82.120,A -90.000,B 90.000,C 0.000} C_DIS
LIN {X -80.273,Y -11.499,Z -81.621,A -90.000,B 90.000,C 0.000} C_DIS
LIN {X -80.578,Y -11.492,Z -81.427,A -90.000,B 90.000,C 0.000} C_DIS
LIN {X -80.996,Y -11.480,Z -81.150,A -90.000,B 90.000,C 0.000} C_DIS
LIN {X -81.790,Y -11.468,Z -80.603,A -90.000,B 90.000,C 0.000} C_DIS
LIN {X -81.963,Y -11.464,Z -80.485,A -90.000,B 90.000,C 0.000} C_DIS
LIN {X -82.182,Y -11.457,Z -80.331,A -90.000,B 90.000,C 0.000} C_DIS
LIN {X -82.291,Y -11.452,Z -80.250,A -90.000,B 90.000,C 0.000} C_DIS
LIN {X -82.683,Y -11.443,Z -79.957,A -90.000,B 90.000,C 0.000} C_DIS
LIN {X -83.257,Y -11.437,Z -79.523,A -90.000,B 90.000,C 0.000} C_DIS
LIN {X -83.641,Y -11.428,Z -79.221,A -90.000,B 90.000,C 0.000} C_DIS
LIN {X -83.832,Y -11.420,Z -79.063,A -90.000,B 90.000,C 0.000} C_DIS
LIN {X -84.624,Y -11.410,Z -78.398,A -90.000,B 90.000,C 0.000} C_DIS
LIN {X -85.201,Y -11.402,Z -77.894,A -90.000,B 90.000,C 0.000} C_DIS
LIN {X -85.697,Y -11.401,Z -77.461,A -90.000,B 90.000,C 0.000} C_DIS
LIN {X -86.474,Y -11.402,Z -76.789,A -90.000,B 90.000,C 0.000} C_DIS
LIN {X -87.053,Y -11.412,Z -76.328,A -90.000,B 90.000,C 0.000} C_DIS
LIN {X -87.600,Y -11.431,Z -75.954,A -90.000,B 90.000,C 0.000} C_DIS
LIN {X -87.774,Y -11.432,Z -75.839,A -90.000,B 90.000,C 0.000} C_DIS
LIN {X -88.193,Y -11.445,Z -75.591,A -90.000,B 90.000,C 0.000} C_DIS
LIN {X -88.534,Y -11.447,Z -75.394,A -90.000,B 90.000,C 0.000} C_DIS
LIN {X -88.748,Y -11.452,Z -75.284,A -90.000,B 90.000,C 0.000} C_DIS
LIN {X -88.944,Y -11.457,Z -75.182,A -90.000,B 90.000,C 0.000} C_DIS
LIN {X -89.082,Y -11.457,Z -75.113,A -90.000,B 90.000,C 0.000} C_DIS
LIN {X -89.518,Y -11.466,Z -74.913,A -90.000,B 90.000,C 0.000} C_DIS
LIN {X -89.953,Y -11.467,Z -74.716,A -90.000,B 90.000,C 0.000} C_DIS
LIN {X -90.405,Y -11.474,Z -74.529,A -90.000,B 90.000,C 0.000} C_DIS
LIN {X -90.864,Y -11.482,Z -74.364,A -90.000,B 90.000,C 0.000} C_DIS
LIN {X -91.072,Y -11.482,Z -74.290,A -90.000,B 90.000,C 0.000} C_DIS
LIN {X -91.464,Y -11.487,Z -74.164,A -90.000,B 90.000,C 0.000} C_DIS
LIN {X -91.623,Y -11.487,Z -74.114,A -90.000,B 90.000,C 0.000} C_DIS
LIN {X -91.887,Y -11.491,Z -74.041,A -90.000,B 90.000,C 0.000} C_DIS
LIN {X -92.088,Y -11.498,Z -73.995,A -90.000,B 90.000,C 0.000} C_DIS
LIN {X -92.510,Y -11.520,Z -73.914,A -90.000,B 90.000,C 0.000} C_DIS
LIN {X -92.630,Y -11.525,Z -73.888,A -90.000,B 90.000,C 0.000} C_DIS
LIN {X -92.748,Y -11.530,Z -73.870,A -90.000,B 90.000,C 0.000} C_DIS
LIN {X -92.951,Y -11.537,Z -73.839,A -90.000,B 90.000,C 0.000} C_DIS
LIN {X -93.235,Y -11.552,Z -73.793,A -90.000,B 90.000,C 0.000} C_DIS
LIN {X -93.459,Y -11.568,Z -73.767,A -90.000,B 90.000,C 0.000} C_DIS
LIN {X -94.120,Y -11.583,Z -73.673,A -90.000,B 90.000,C 0.000} C_DIS
